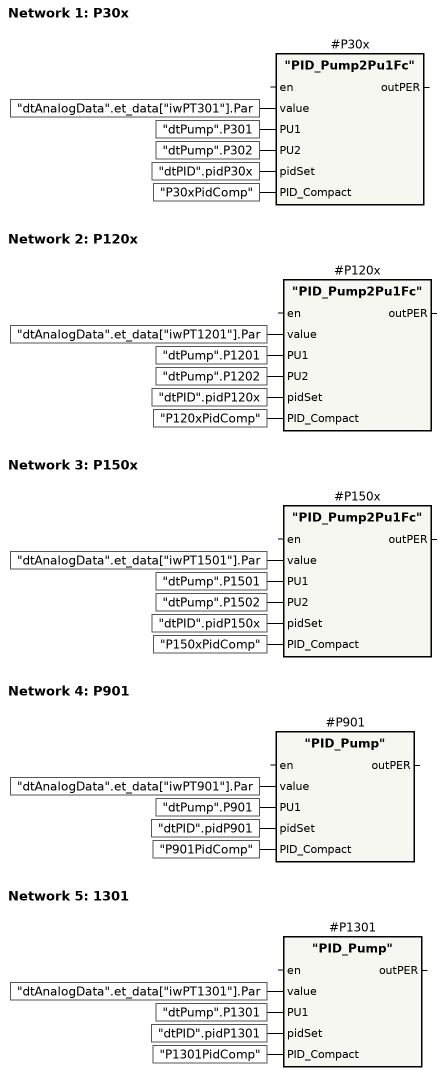
   #P30x(value := "dtAnalogData".et_data["iwPT301"].Par,   // "PID_Pump2Pu1Fc"
         PU1 := "dtPump".P301,
         PU2 := "dtPump".P302,
         pidSet := "dtPID".pidP30x,
         PID_Compact := "P30xPidComp");
END_REGION

REGION Network 2: P120x
   #P120x(value := "dtAnalogData".et_data["iwPT1201"].Par,   // "PID_Pump2Pu1Fc"
          PU1 := "dtPump".P1201,
          PU2 := "dtPump".P1202,
          pidSet := "dtPID".pidP120x,
          PID_Compact := "P120xPidComp");
END_REGION

REGION Network 3: P150x
   #P150x(value := "dtAnalogData".et_data["iwPT1501"].Par,   // "PID_Pump2Pu1Fc"
          PU1 := "dtPump".P1501,
          PU2 := "dtPump".P1502,
          pidSet := "dtPID".pidP150x,
          PID_Compact := "P150xPidComp");
END_REGION

REGION Network 4: P901
   #P901(value := "dtAnalogData".et_data["iwPT901"].Par,   // "PID_Pump"
         PU1 := "dtPump".P901,
         pidSet := "dtPID".pidP901,
         PID_Compact := "P901PidComp");
END_REGION

REGION Network 5: 1301
   #P1301(value := "dtAnalogData".et_data["iwPT1301"].Par,   // "PID_Pump"
          PU1 := "dtPump".P1301,
          pidSet := "dtPID".pidP1301,
          PID_Compact := "P1301PidComp");
END_REGION
END_FUNCTION_BLOCK

FUNCTION_BLOCK "PID_Pump2Pu1Fc"   // FB59, FBD
{ S7_Optimized_Access := 'TRUE' }
VERSION : 0.1
// stored: AutoNumber true, IsIECCheckEnabled false, IsRetainMemResEnabled false, MemoryReserve 100, SetENOAutomatically false, UDAEnableTagReadback false
   VAR_INPUT
      value : Real;
      PU1 : "Pump";
      PU2 : "Pump";
   END_VAR
   VAR_OUTPUT
      outPER : Int;
   END_VAR
   VAR_IN_OUT
      pidSet : "setPID";
      PID_Compact : PID_Compact;
   END_VAR
   VAR
      pTrigAutoMode : Bool;
      pTrigManualMode : Bool;
      pTrigCmAuto1 : Bool;
      pTrigCmAuto2 : Bool;
      nTrigCmAuto1 : Bool;
      nTrigCmAuto2 : Bool;
      pTrigFix : Bool;
      nTrigFix : Bool;
      pTrigFreez : Bool;
      nTrigFreez : Bool;
      pTrigCmHand : Bool;
      nTrigCmHand : Bool;
   END_VAR
   VAR_TEMP   // added for the SCL form of the ladder/FBD networks
      _w1 : Bool;
      _w2 : Bool;
      _w3 : Bool;
      _w4 : Bool;
      _w5 : Bool;
      _w6 : Bool;
      _w7 : Bool;
      _w8 : Bool;
      _w9 : Bool;
      _w10 : Bool;
   END_VAR
BEGIN

REGION Network 1: Интеграл
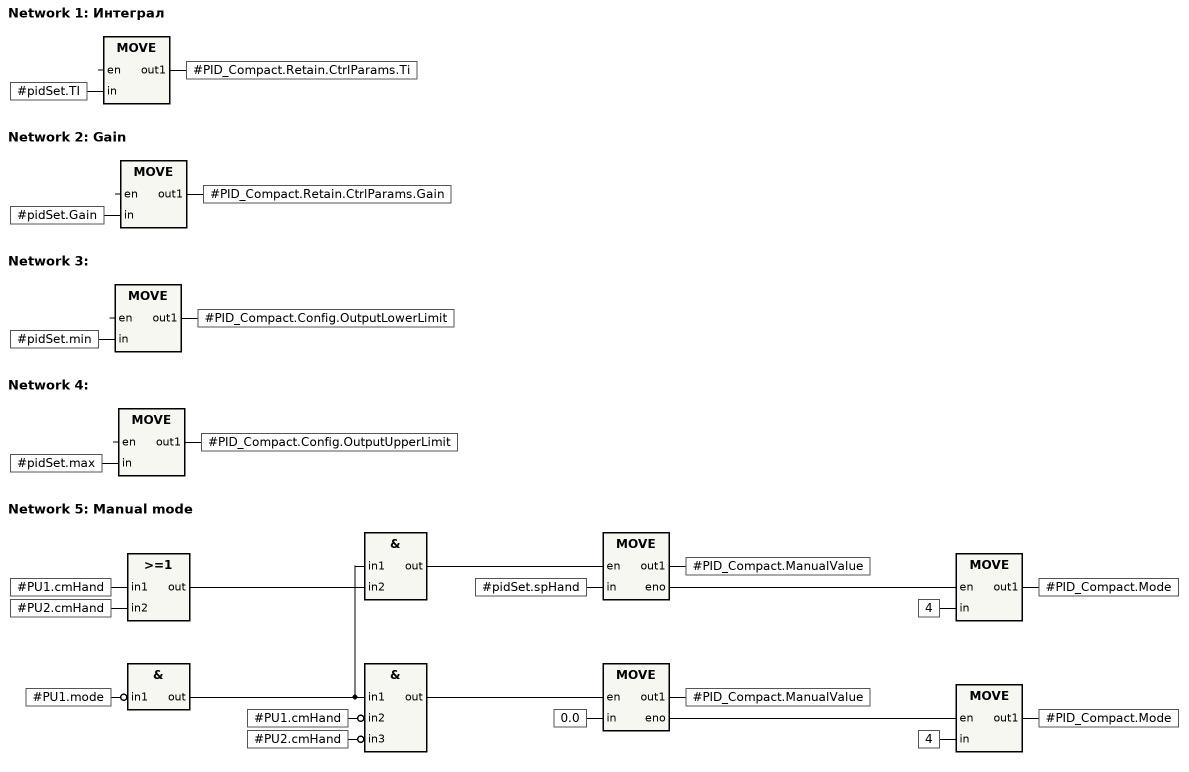
   #PID_Compact.Retain.CtrlParams.Ti := #pidSet.TI;
END_REGION

REGION Network 2: Gain
   #PID_Compact.Retain.CtrlParams.Gain := #pidSet.Gain;
END_REGION

REGION Network 3
   #PID_Compact.Config.OutputLowerLimit := #pidSet.min;
END_REGION

REGION Network 4
   #PID_Compact.Config.OutputUpperLimit := #pidSet.max;
END_REGION

REGION Network 5: Manual mode
   IF NOT #PU1.mode AND (#PU1.cmHand OR #PU2.cmHand) THEN
       #PID_Compact.ManualValue := #pidSet.spHand;
       #PID_Compact.Mode := 4;
   END_IF;
   IF NOT #PU1.mode AND NOT #PU1.cmHand AND NOT #PU2.cmHand THEN
       #PID_Compact.ManualValue := 0.0;
       #PID_Compact.Mode := 4;
   END_IF;
END_REGION

REGION Network 6: Auto mode
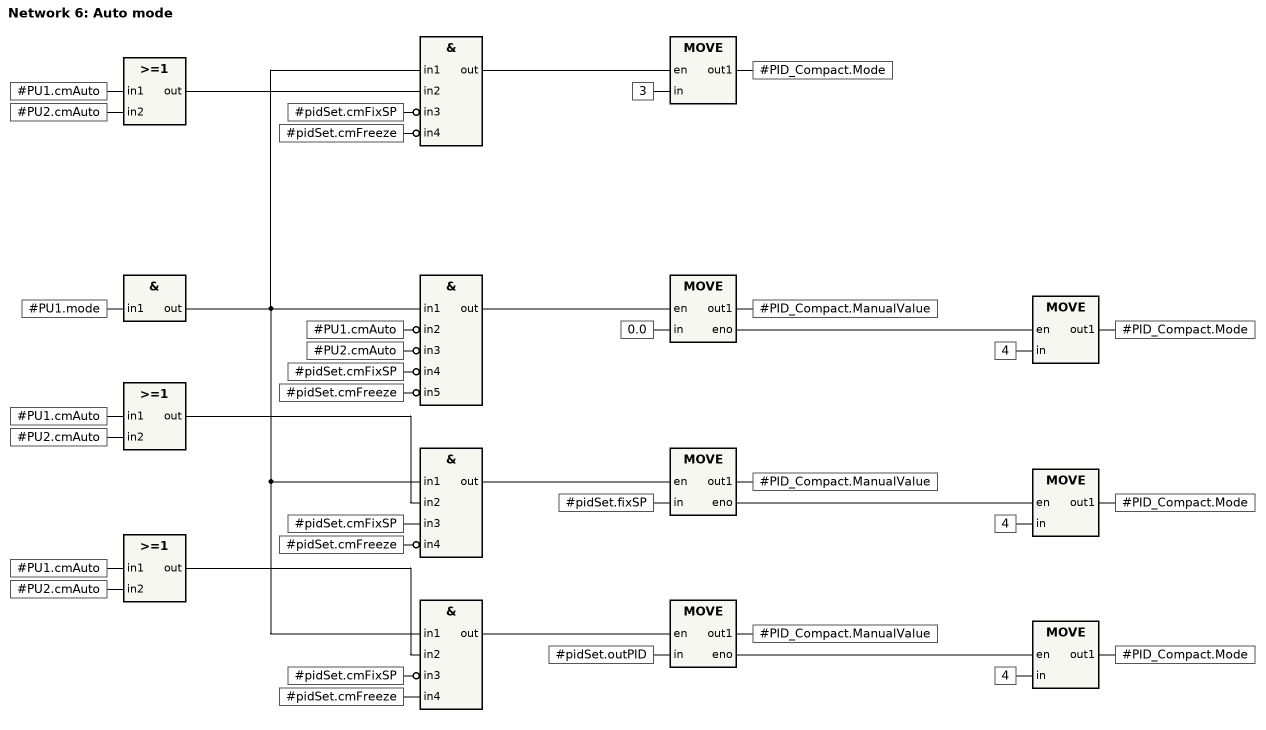
   IF #PU1.mode AND (#PU1.cmAuto OR #PU2.cmAuto) AND NOT #pidSet.cmFixSP AND NOT #pidSet.cmFreeze THEN
       #PID_Compact.Mode := 3;
   END_IF;
   IF #PU1.mode AND NOT #PU1.cmAuto AND NOT #PU2.cmAuto AND NOT #pidSet.cmFixSP AND NOT #pidSet.cmFreeze THEN
       #PID_Compact.ManualValue := 0.0;
       #PID_Compact.Mode := 4;
   END_IF;
   IF #PU1.mode AND (#PU1.cmAuto OR #PU2.cmAuto) AND #pidSet.cmFixSP AND NOT #pidSet.cmFreeze THEN
       #PID_Compact.ManualValue := #pidSet.fixSP;
       #PID_Compact.Mode := 4;
   END_IF;
   IF #PU1.mode AND (#PU1.cmAuto OR #PU2.cmAuto) AND NOT #pidSet.cmFixSP AND #pidSet.cmFreeze THEN
       #PID_Compact.ManualValue := #pidSet.outPID;
       #PID_Compact.Mode := 4;
   END_IF;
END_REGION

REGION Network 7: Set modeActivate
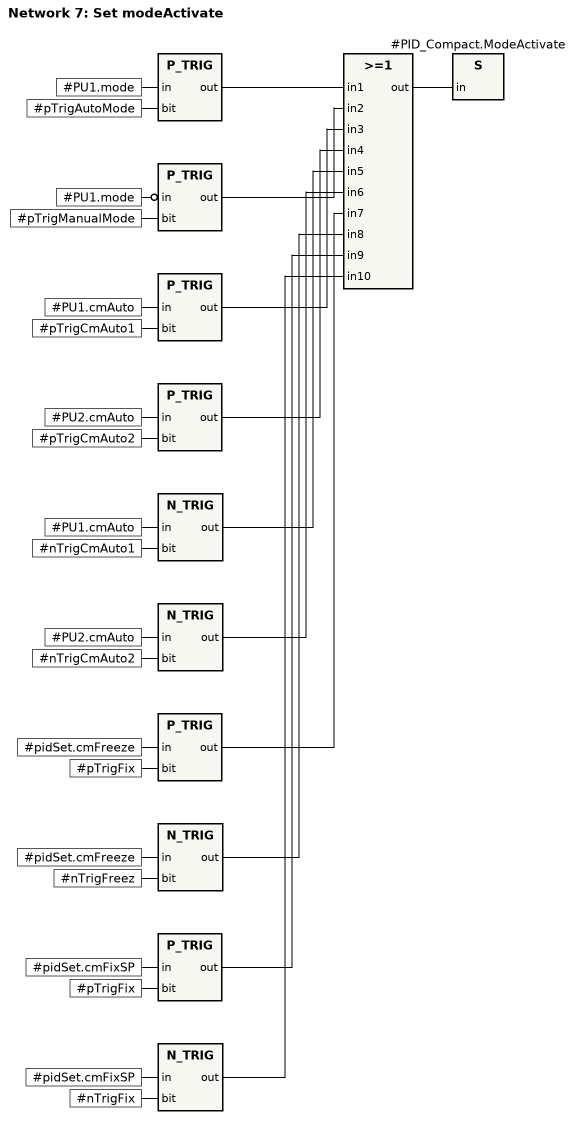
   #_w1 := #PU1.mode AND NOT #pTrigAutoMode;   // rising edge
   #pTrigAutoMode := #PU1.mode;
   #_w2 := NOT #PU1.mode AND NOT #pTrigManualMode;   // rising edge
   #pTrigManualMode := NOT #PU1.mode;
   #_w3 := #PU1.cmAuto AND NOT #pTrigCmAuto1;   // rising edge
   #pTrigCmAuto1 := #PU1.cmAuto;
   #_w4 := #PU2.cmAuto AND NOT #pTrigCmAuto2;   // rising edge
   #pTrigCmAuto2 := #PU2.cmAuto;
   #_w5 := NOT #PU1.cmAuto AND #nTrigCmAuto1;   // falling edge
   #nTrigCmAuto1 := #PU1.cmAuto;
   #_w6 := NOT #PU2.cmAuto AND #nTrigCmAuto2;   // falling edge
   #nTrigCmAuto2 := #PU2.cmAuto;
   #_w7 := #pidSet.cmFreeze AND NOT #pTrigFix;   // rising edge
   #pTrigFix := #pidSet.cmFreeze;
   #_w8 := NOT #pidSet.cmFreeze AND #nTrigFreez;   // falling edge
   #nTrigFreez := #pidSet.cmFreeze;
   #_w9 := #pidSet.cmFixSP AND NOT #pTrigFix;   // rising edge
   #pTrigFix := #pidSet.cmFixSP;
   #_w10 := NOT #pidSet.cmFixSP AND #nTrigFix;   // falling edge
   #nTrigFix := #pidSet.cmFixSP;
   IF #_w1 OR #_w2 OR #_w3 OR #_w4 OR #_w5 OR #_w6 OR #_w7 OR #_w8 OR #_w9 OR #_w10 THEN
       #PID_Compact.ModeActivate := TRUE;
   END_IF;
END_REGION

REGION Network 8
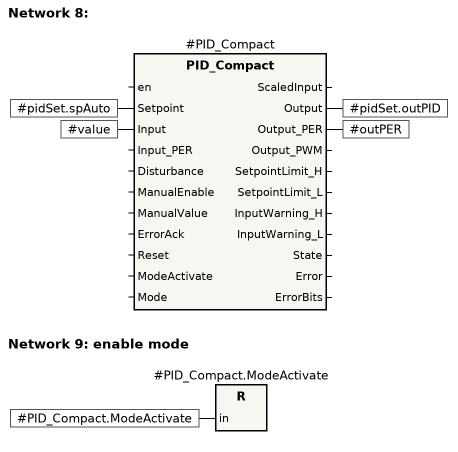
   #PID_Compact(Setpoint := #pidSet.spAuto, Input := #value, Output => #pidSet.outPID, Output_PER => #outPER);   // PID_Compact
END_REGION

REGION Network 9: enable mode
   IF #PID_Compact.ModeActivate THEN #PID_Compact.ModeActivate := FALSE; END_IF;
END_REGION
END_FUNCTION_BLOCK

FUNCTION_BLOCK "PID_Pump"   // FB62, FBD
{ S7_Optimized_Access := 'TRUE' }
VERSION : 0.1
// stored: AutoNumber false, IsIECCheckEnabled false, IsRetainMemResEnabled false, MemoryReserve 100, SetENOAutomatically false, UDAEnableTagReadback false
   VAR_INPUT
      value : Real;
      PU1 : "Pump";
   END_VAR
   VAR_OUTPUT
      outPER : Int;
   END_VAR
   VAR_IN_OUT
      pidSet : "setPID";
      PID_Compact : PID_Compact;
   END_VAR
   VAR
      pTrigAutoMode : Bool;
      pTrigManualMode : Bool;
      pTrigCmAuto1 : Bool;
      pTrigCmAuto2 : Bool;
      nTrigCmAuto1 : Bool;
      nTrigCmAuto2 : Bool;
      pTrigFix : Bool;
      nTrigFix : Bool;
      pTrigFreez : Bool;
      nTrigFreez : Bool;
      pTrigCmHand : Bool;
      nTrigCmHand : Bool;
   END_VAR
   VAR_TEMP   // added for the SCL form of the ladder/FBD networks
      _w1 : Bool;
      _w2 : Bool;
      _w3 : Bool;
      _w4 : Bool;
      _w5 : Bool;
      _w6 : Bool;
      _w7 : Bool;
      _w8 : Bool;
   END_VAR
BEGIN

REGION Network 1: Интеграл
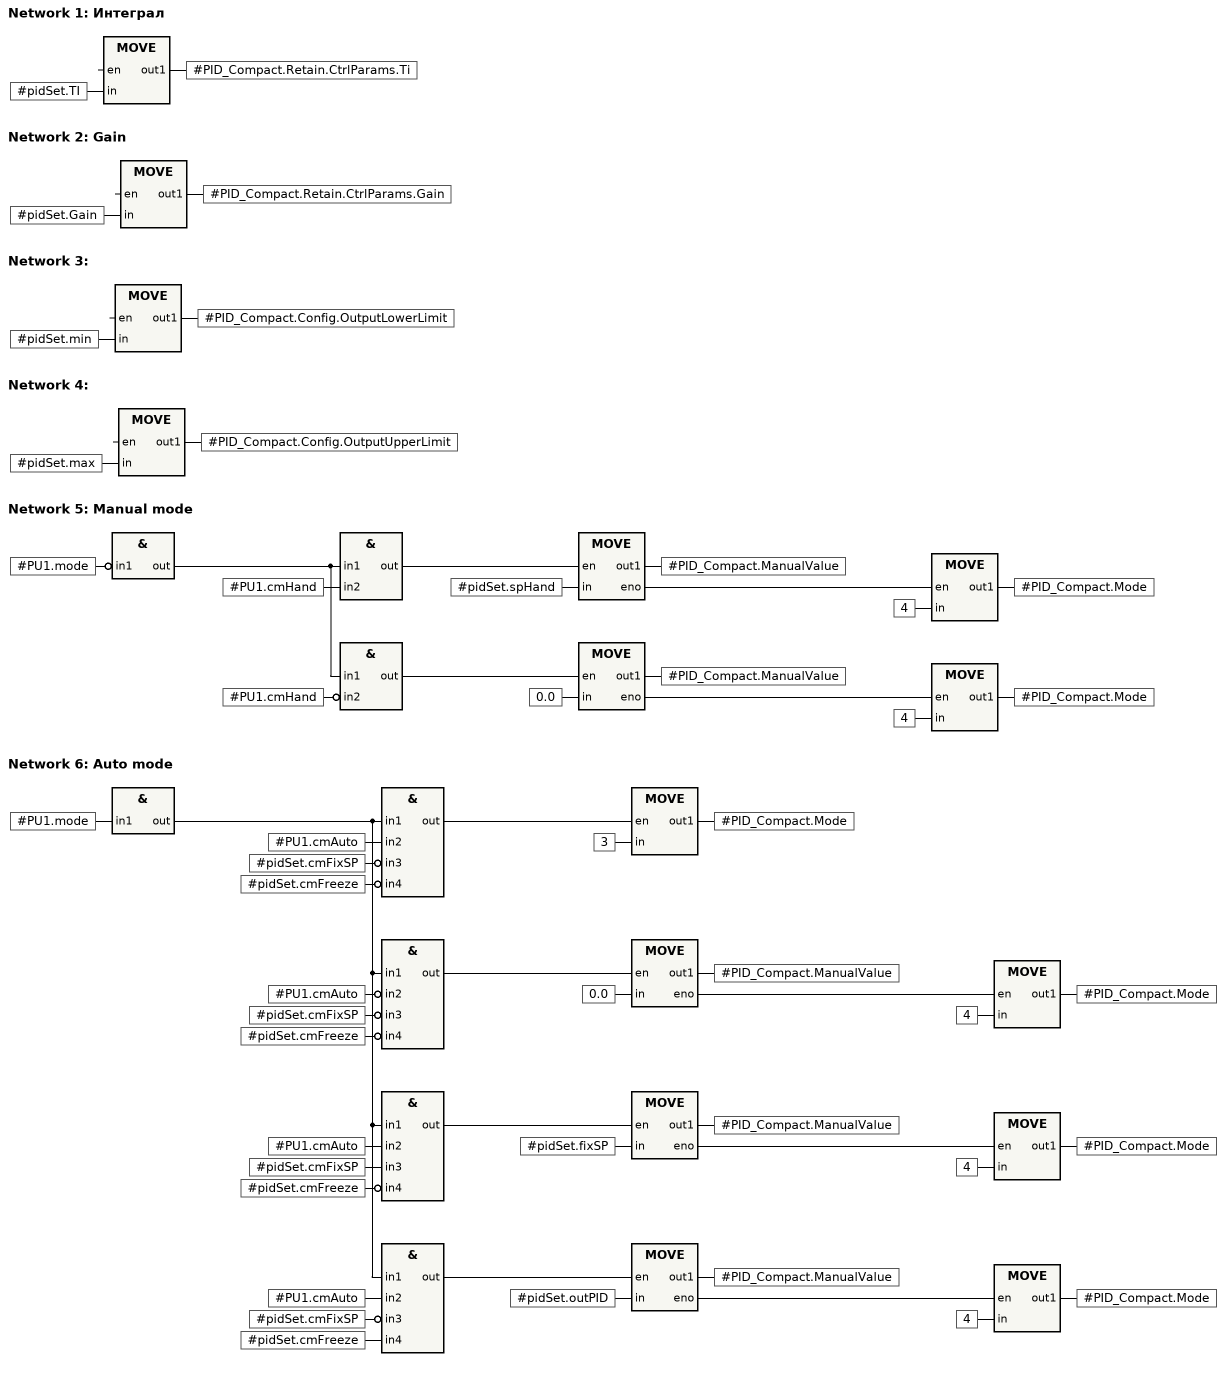
   #PID_Compact.Retain.CtrlParams.Ti := #pidSet.TI;
END_REGION

REGION Network 2: Gain
   #PID_Compact.Retain.CtrlParams.Gain := #pidSet.Gain;
END_REGION

REGION Network 3
   #PID_Compact.Config.OutputLowerLimit := #pidSet.min;
END_REGION

REGION Network 4
   #PID_Compact.Config.OutputUpperLimit := #pidSet.max;
END_REGION

REGION Network 5: Manual mode
   IF NOT #PU1.mode AND #PU1.cmHand THEN
       #PID_Compact.ManualValue := #pidSet.spHand;
       #PID_Compact.Mode := 4;
   END_IF;
   IF NOT #PU1.mode AND NOT #PU1.cmHand THEN
       #PID_Compact.ManualValue := 0.0;
       #PID_Compact.Mode := 4;
   END_IF;
END_REGION

REGION Network 6: Auto mode
   IF #PU1.mode AND #PU1.cmAuto AND NOT #pidSet.cmFixSP AND NOT #pidSet.cmFreeze THEN
       #PID_Compact.Mode := 3;
   END_IF;
   IF #PU1.mode AND NOT #PU1.cmAuto AND NOT #pidSet.cmFixSP AND NOT #pidSet.cmFreeze THEN
       #PID_Compact.ManualValue := 0.0;
       #PID_Compact.Mode := 4;
   END_IF;
   IF #PU1.mode AND #PU1.cmAuto AND #pidSet.cmFixSP AND NOT #pidSet.cmFreeze THEN
       #PID_Compact.ManualValue := #pidSet.fixSP;
       #PID_Compact.Mode := 4;
   END_IF;
   IF #PU1.mode AND #PU1.cmAuto AND NOT #pidSet.cmFixSP AND #pidSet.cmFreeze THEN
       #PID_Compact.ManualValue := #pidSet.outPID;
       #PID_Compact.Mode := 4;
   END_IF;
END_REGION

REGION Network 7: Set modeActivate
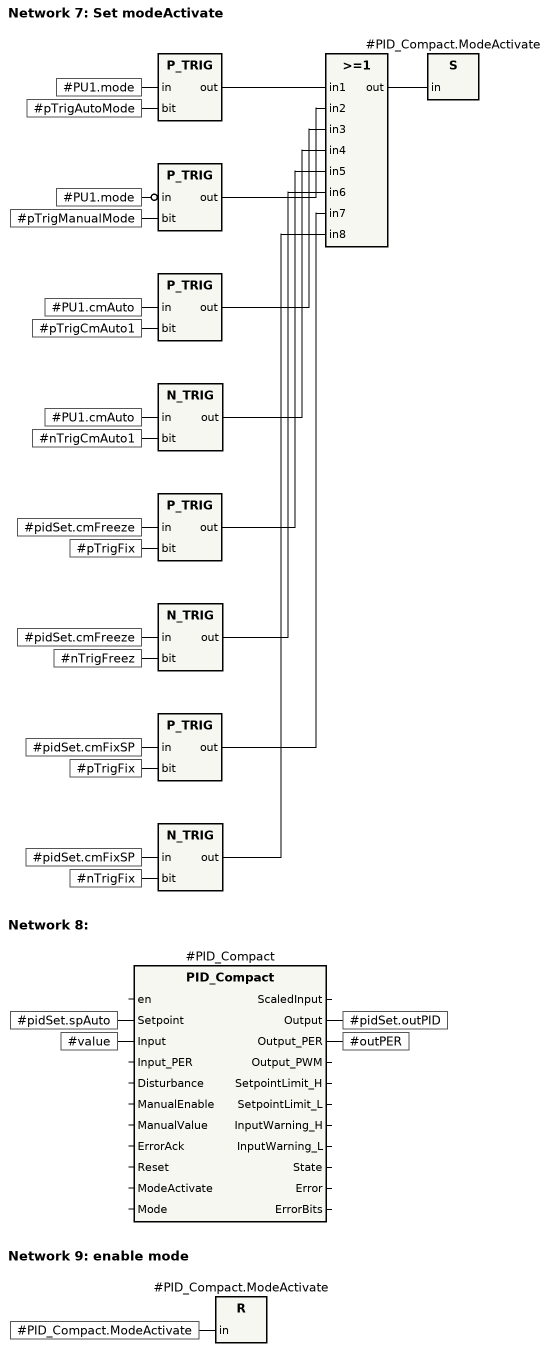
   #_w1 := #PU1.mode AND NOT #pTrigAutoMode;   // rising edge
   #pTrigAutoMode := #PU1.mode;
   #_w2 := NOT #PU1.mode AND NOT #pTrigManualMode;   // rising edge
   #pTrigManualMode := NOT #PU1.mode;
   #_w3 := #PU1.cmAuto AND NOT #pTrigCmAuto1;   // rising edge
   #pTrigCmAuto1 := #PU1.cmAuto;
   #_w4 := NOT #PU1.cmAuto AND #nTrigCmAuto1;   // falling edge
   #nTrigCmAuto1 := #PU1.cmAuto;
   #_w5 := #pidSet.cmFreeze AND NOT #pTrigFix;   // rising edge
   #pTrigFix := #pidSet.cmFreeze;
   #_w6 := NOT #pidSet.cmFreeze AND #nTrigFreez;   // falling edge
   #nTrigFreez := #pidSet.cmFreeze;
   #_w7 := #pidSet.cmFixSP AND NOT #pTrigFix;   // rising edge
   #pTrigFix := #pidSet.cmFixSP;
   #_w8 := NOT #pidSet.cmFixSP AND #nTrigFix;   // falling edge
   #nTrigFix := #pidSet.cmFixSP;
   IF #_w1 OR #_w2 OR #_w3 OR #_w4 OR #_w5 OR #_w6 OR #_w7 OR #_w8 THEN
       #PID_Compact.ModeActivate := TRUE;
   END_IF;
END_REGION

REGION Network 8
   #PID_Compact(Setpoint := #pidSet.spAuto, Input := #value, Output => #pidSet.outPID, Output_PER => #outPER);   // PID_Compact
END_REGION

REGION Network 9: enable mode
   IF #PID_Compact.ModeActivate THEN #PID_Compact.ModeActivate := FALSE; END_IF;
END_REGION
END_FUNCTION_BLOCK

FUNCTION_BLOCK "TONR_200ms"   // FB10, FBD
{ S7_Optimized_Access := 'TRUE' }
VERSION : 0.1
// stored: AutoNumber true, IsIECCheckEnabled false, IsRetainMemResEnabled false, MemoryReserve 100, SetENOAutomatically false, UDAEnableTagReadback false
   VAR_INPUT
      In : Bool;
      PT : Time;
      R : Bool;
   END_VAR
   VAR_OUTPUT
      ET : Time;
      Q : Bool;
   END_VAR
BEGIN

REGION Network 1: Увеличение текущего времени
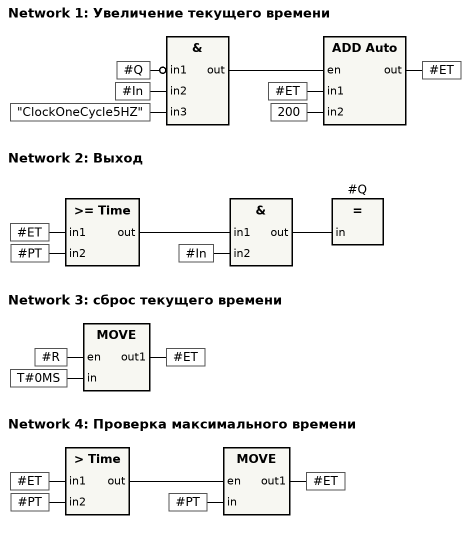
   IF NOT #Q AND #In AND "ClockOneCycle5HZ" THEN #ET := #ET + 200; END_IF;
END_REGION

REGION Network 2: Выход
   #Q := (#ET >= #PT) AND #In;
END_REGION

REGION Network 3: сброс текущего времени
   IF #R THEN #ET := T#0MS; END_IF;
END_REGION

REGION Network 4: Проверка максимального времени
   IF #ET > #PT THEN #ET := #PT; END_IF;
END_REGION
END_FUNCTION_BLOCK

FUNCTION_BLOCK "TON_200ms"   // FB9, FBD
{ S7_Optimized_Access := 'TRUE' }
VERSION : 0.1
// stored: AutoNumber true, IsIECCheckEnabled false, IsRetainMemResEnabled false, MemoryReserve 100, SetENOAutomatically false, UDAEnableTagReadback false
   VAR_INPUT
      In : Bool;
      PT : Time;
   END_VAR
   VAR_OUTPUT
      ET : Time;
      Q : Bool;
   END_VAR
BEGIN

REGION Network 1: Увеличение текущего времени
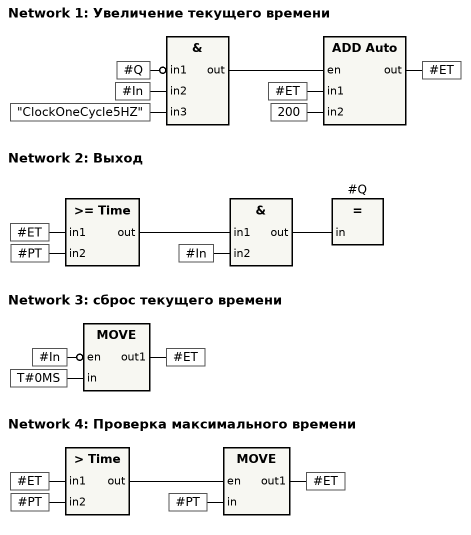
   IF NOT #Q AND #In AND "ClockOneCycle5HZ" THEN #ET := #ET + 200; END_IF;
END_REGION

REGION Network 2: Выход
   #Q := (#ET >= #PT) AND #In;
END_REGION

REGION Network 3: сброс текущего времени
   IF NOT #In THEN #ET := T#0MS; END_IF;
END_REGION

REGION Network 4: Проверка максимального времени
   IF #ET > #PT THEN #ET := #PT; END_IF;
END_REGION
END_FUNCTION_BLOCK

FUNCTION "setFlags" : Void   // FC2, FBD
{ S7_Optimized_Access := 'TRUE' }
VERSION : 0.1
// stored: AutoNumber true, IsIECCheckEnabled false, SetENOAutomatically false, UDAEnableTagReadback false
   VAR_INPUT
      enCondition : Bool;
      condition : Bool;
      setTimerVal : Real;
   END_VAR
   VAR_IN_OUT
      curFlag : Bool;
      mainFlag : Bool;
      timerVal : Real;
   END_VAR
BEGIN

REGION Network 1 (SCL)

   #curFlag := #enCondition AND #condition;

   IF NOT #curFlag THEN
       #timerVal := 0;
   END_IF;

   IF #curFlag AND #timerVal < #setTimerVal THEN
       #timerVal += 0.1;
   END_IF;

   IF #timerVal >= #setTimerVal THEN
       #mainFlag := TRUE;
   END_IF;
END_REGION
END_FUNCTION

FUNCTION "setState" : Void   // FC3, FBD
{ S7_Optimized_Access := 'TRUE' }
VERSION : 0.1
// stored: AutoNumber true, IsIECCheckEnabled false, SetENOAutomatically false, UDAEnableTagReadback false
   VAR_INPUT
      condition : Bool;
      hexVal : Word;
   END_VAR
   VAR_IN_OUT
      state : Word;
   END_VAR
BEGIN

REGION Network 1 (SCL)
   IF #condition THEN
       // Statement section IF
       #state := #state OR #hexVal;
   ELSE
       #state := #state AND NOT #hexVal;
   END_IF;
END_REGION
END_FUNCTION

FUNCTION_BLOCK "DPumpCntr"   // FB70, LAD
{ S7_Optimized_Access := 'FALSE' }
VERSION : 0.1
// #ST:
// номер бита, часло десятичное
//  0  - стоп 
// 0 1 - работа
// 1 2 - запуск
// 2 4 - остановка
// 3 8 - сервисный режим
// 4 16 - ошибка Пуска
// 5 32 - ошибка Стопа
// 6 64 - ошибка питания
// 7 128 - ошибка частотника (дозатора)
// 8 256 - Блокировка внешняя
// 9 - 512 - нажат аварийный стоп
// 10 -1024 - сборная авария
// 11 2048
// 12 4096
// 13 8192
// 14 16384 
// 15 32768 - режим 0-ручной, 1-авто
// 
// показывать кнопки ручного управления
// stored: AutoNumber false, IsIECCheckEnabled false, SetENOAutomatically false, UDAEnableTagReadback false
   VAR_INPUT
      power : Bool;   // питание устройства
      run : Bool;
      emrStop : Bool;   // Авариный стоп 0-авария, 1-ок
      alarmFC : Bool;   // 1-авария
      Ack : Bool;   // Сброс Аварий
      FE : Real;
   END_VAR
   VAR_OUTPUT
      qStart : Bool;
      pqw : Int;
   END_VAR
   VAR_IN_OUT
      dev : "DPump";
      prop : "PropDosing";
   END_VAR
   VAR DB_SPECIFIC
      ErrOC : Bool;   // Признак аварии по закрытию или открытию
      ErrPower : Bool;   // Признак аварии питания
      ErrDis : Bool;   // Признак внешней блокировки
      qON : Bool;   // Выход для управления механизмом
      tmrClosing { S7_SetPoint := 'True'} : TON_TIME;
      tmrOpening { S7_SetPoint := 'True'} : TON_TIME;
      closed : Bool;
      opened : Bool;
      closing : Bool;
      opening : Bool;
      errStart : Bool;
      errStop : Bool;
      errEmrStop : Bool;
      errAlarmFc : Bool;
      errService : Bool;
      tStart : Time;
      tStop : Time;
   END_VAR
   VAR
      ServiceEventHandler { S7_SetPoint := 'True'} : "DevAckSingleAlarm";
      PowerEventHandler { S7_SetPoint := 'True'} : "DevAckSingleAlarm";
      DevAlarmEventHandler { S7_SetPoint := 'True'} : "DevAckSingleAlarm";
      DisEventHandler { S7_SetPoint := 'True'} : "DevAckSingleAlarm";
      EmrStopEventHandler { S7_SetPoint := 'True'} : "DevAckSingleAlarm";
      BadStartEventHandler { S7_SetPoint := 'True'} : "DevAckSingleAlarm";
      BadStopEventHandler { S7_SetPoint := 'True'} : "DevAckSingleAlarm";
   END_VAR
BEGIN

REGION Network 1: Сброс состояния
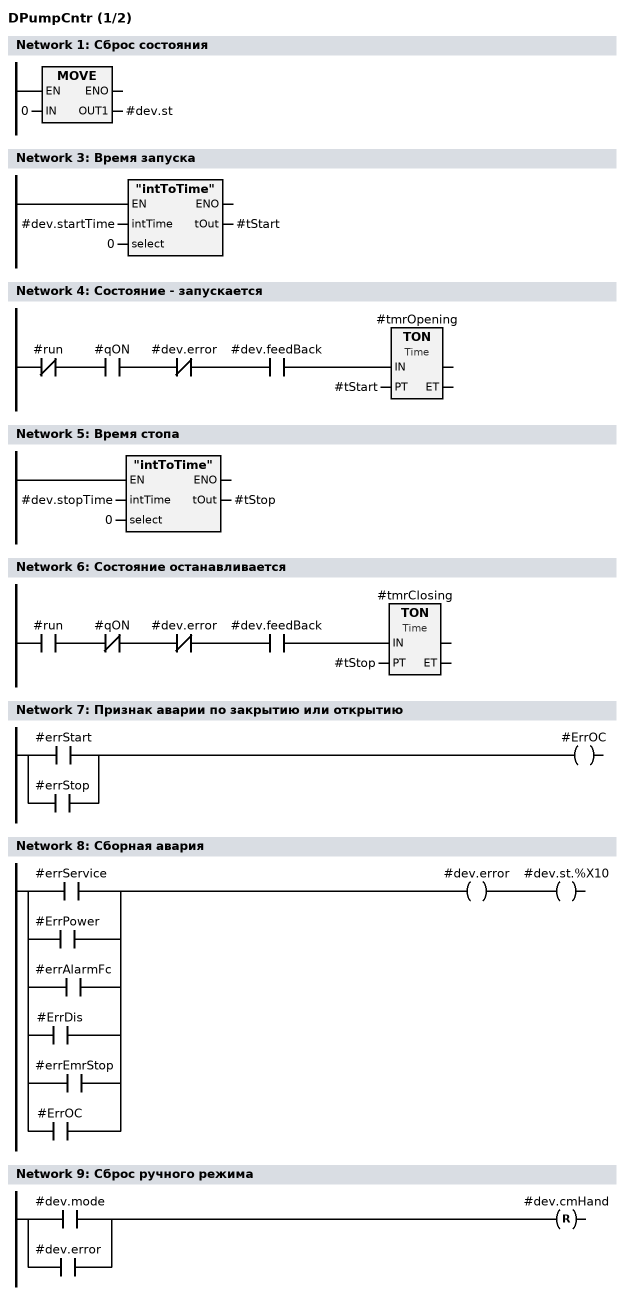
   RUNG wire#powerrail
      { S7_GenerateENO := "TRUE" } Move(in := 0, out1 => #dev.st)
   END_RUNG
   // the same network as SCL:
   #dev.st := 0;
END_REGION

REGION Network 2 (SCL): Event handlers
   #ServiceEventHandler(alarmSignal := #dev.service,
                        ack := #Ack,
                        ackBit := #dev.ack.%X3,
                        stateBit := #dev.st.%X3,
                        alarmTag := #errService);
   #BadStartEventHandler(alarmSignal:=#tmrOpening.Q,
                         ack:=#Ack,
                         ackBit:=#dev.ack.%X4,
                         stateBit:=#dev.st.%X4,
                         alarmTag:=#errStart);
   #BadStopEventHandler(alarmSignal:=#tmrClosing.Q,
                        ack:=#Ack,
                        ackBit:=#dev.ack.%X5,
                        stateBit:=#dev.ack.%X5,
                        alarmTag:=#errStop);
   #PowerEventHandler(alarmSignal := #power,
                      ack := #Ack,
                      ackBit := #dev.ack.%X6,
                      stateBit := #dev.st.%X6,
                      alarmTag := #ErrPower);
   #DevAlarmEventHandler(alarmSignal := #alarmFC,
                         ack := #Ack,
                         ackBit := #dev.ack.%X7,
                         stateBit := #dev.st.%X7,
                         alarmTag := #errAlarmFc);
   #DisEventHandler(alarmSignal := #dev.block,
                    ack := #Ack,
                    ackBit := #dev.ack.%X8,
                    stateBit := #dev.st.%X8,
                    alarmTag := #ErrDis);
   #EmrStopEventHandler(alarmSignal := #emrStop,
                        ack := #Ack,
                        ackBit := #dev.ack.%X9,
                        stateBit := #dev.st.%X9,
                        alarmTag := #errEmrStop);
END_REGION

REGION Network 3: Время запуска
   RUNG wire#powerrail
      "intToTime"(intTime := #dev.startTime, select := 0, tOut => #tStart)
   END_RUNG
   // the same network as SCL:
   "intToTime"(intTime := #dev.startTime, select := 0, tOut => #tStart);
END_REGION

REGION Network 4: Состояние - запускается
   RUNG wire#powerrail
      I_Contact( #run )
      Contact( #qON )
      I_Contact( #dev.error )
      Contact( #dev.feedBack )
      { S7_Templates := "time_type := Time" } #tmrOpening.TON(pt := #tStart, et =>)
   END_RUNG
   // the same network as SCL:
   #tmrOpening(IN := NOT #run AND #qON AND NOT #dev.error AND #dev.feedBack, PT := #tStart);   // TON
END_REGION

REGION Network 5: Время стопа
   RUNG wire#powerrail
      "intToTime"(intTime := #dev.stopTime, select := 0, tOut => #tStop)
   END_RUNG
   // the same network as SCL:
   "intToTime"(intTime := #dev.stopTime, select := 0, tOut => #tStop);
END_REGION

REGION Network 6: Состояние останавливается
   RUNG wire#powerrail
      Contact( #run )
      I_Contact( #qON )
      I_Contact( #dev.error )
      Contact( #dev.feedBack )
      { S7_Templates := "time_type := Time" } #tmrClosing.TON(pt := #tStop, et =>)
   END_RUNG
   // the same network as SCL:
   #tmrClosing(IN := #run AND NOT #qON AND NOT #dev.error AND #dev.feedBack, PT := #tStop);   // TON
END_REGION

REGION Network 7: Признак аварии по закрытию или открытию
   RUNG wire#powerrail
      Contact( #errStart )
      wire#w1
      Coil( #ErrOC )
   END_RUNG
   RUNG wire#powerrail
      Contact( #errStop )
   END_RUNG wire#w1
   // the same network as SCL:
   #ErrOC := #errStart OR #errStop;
END_REGION

REGION Network 8: Сборная авария
   RUNG wire#powerrail
      Contact( #errService )
      wire#w1
      Coil( #dev.error )
      Coil( #dev.st.%X10 )
   END_RUNG
   RUNG wire#powerrail
      Contact( #ErrPower )
   END_RUNG wire#w1
   RUNG wire#powerrail
      Contact( #errAlarmFc )
   END_RUNG wire#w1
   RUNG wire#powerrail
      Contact( #ErrDis )
   END_RUNG wire#w1
   RUNG wire#powerrail
      Contact( #errEmrStop )
   END_RUNG wire#w1
   RUNG wire#powerrail
      Contact( #ErrOC )
   END_RUNG wire#w1
   // the same network as SCL:
   #dev.error := #errService OR #ErrPower OR #errAlarmFc OR #ErrDis OR #errEmrStop OR #ErrOC;
   #dev.st.%X10 := #dev.error;
END_REGION

REGION Network 9: Сброс ручного режима
   RUNG wire#powerrail
      Contact( #dev.mode )
      wire#w1
      R_Coil( #dev.cmHand )
   END_RUNG
   RUNG wire#powerrail
      Contact( #dev.error )
   END_RUNG wire#w1
   // the same network as SCL:
   IF #dev.mode OR #dev.error THEN #dev.cmHand := FALSE; END_IF;
END_REGION

REGION Network 10: Сброс авто режима
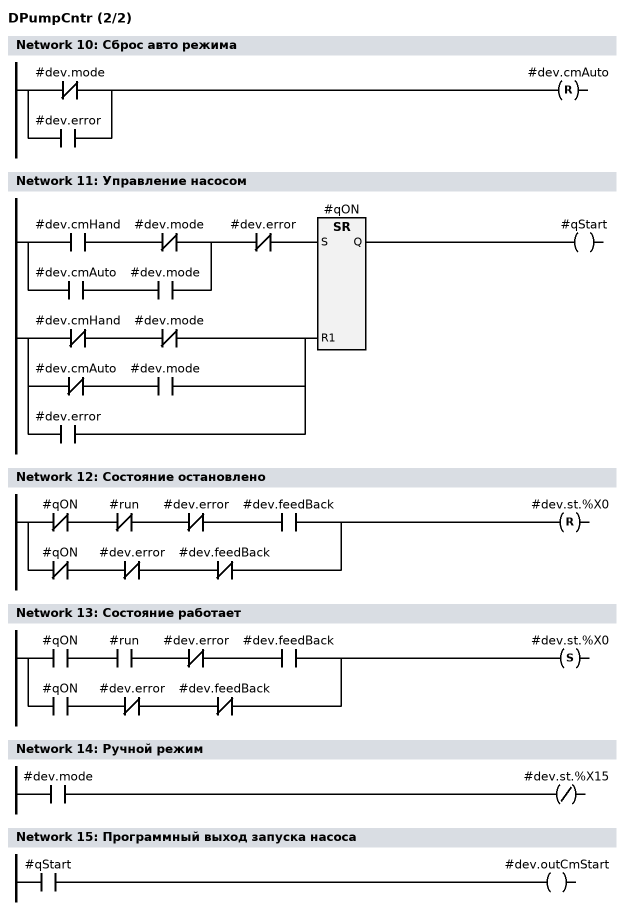
   RUNG wire#powerrail
      I_Contact( #dev.mode )
      wire#w1
      R_Coil( #dev.cmAuto )
   END_RUNG
   RUNG wire#powerrail
      Contact( #dev.error )
   END_RUNG wire#w1
   // the same network as SCL:
   IF NOT #dev.mode OR #dev.error THEN #dev.cmAuto := FALSE; END_IF;
END_REGION

REGION Network 11: Управление насосом
   RUNG wire#powerrail
      Contact( #dev.cmHand )
      I_Contact( #dev.mode )
      wire#w1
      I_Contact( #dev.error )
      S_SR(operand := #qON, r1 := wire#w2)
      Coil( #qStart )
   END_RUNG
   RUNG wire#powerrail
      Contact( #dev.cmAuto )
      Contact( #dev.mode )
   END_RUNG wire#w1
   RUNG wire#powerrail
      I_Contact( #dev.cmHand )
      I_Contact( #dev.mode )
   END_RUNG wire#w2
   RUNG wire#powerrail
      I_Contact( #dev.cmAuto )
      Contact( #dev.mode )
   END_RUNG wire#w2
   RUNG wire#powerrail
      Contact( #dev.error )
   END_RUNG wire#w2
   // the same network as SCL:
   IF ((#dev.cmHand AND NOT #dev.mode) OR (#dev.cmAuto AND #dev.mode)) AND NOT #dev.error THEN
       #qON := TRUE;   // SR flip-flop
   END_IF;
   IF (NOT #dev.cmHand AND NOT #dev.mode) OR (NOT #dev.cmAuto AND #dev.mode) OR #dev.error THEN
       #qON := FALSE;
   END_IF;
   #qStart := #qON;
END_REGION

REGION Network 12: Состояние остановлено
   RUNG wire#powerrail
      I_Contact( #qON )
      I_Contact( #run )
      I_Contact( #dev.error )
      Contact( #dev.feedBack )
      wire#w1
      R_Coil( #dev.st.%X0 )
   END_RUNG
   RUNG wire#powerrail
      I_Contact( #qON )
      I_Contact( #dev.error )
      I_Contact( #dev.feedBack )
   END_RUNG wire#w1
   // the same network as SCL:
   IF (NOT #qON AND NOT #run AND NOT #dev.error AND #dev.feedBack) OR (NOT #qON AND NOT #dev.error AND NOT #dev.feedBack) THEN
       #dev.st.%X0 := FALSE;
   END_IF;
END_REGION

REGION Network 13: Состояние работает
   RUNG wire#powerrail
      Contact( #qON )
      Contact( #run )
      I_Contact( #dev.error )
      Contact( #dev.feedBack )
      wire#w1
      S_Coil( #dev.st.%X0 )
   END_RUNG
   RUNG wire#powerrail
      Contact( #qON )
      I_Contact( #dev.error )
      I_Contact( #dev.feedBack )
   END_RUNG wire#w1
   // the same network as SCL:
   IF (#qON AND #run AND NOT #dev.error AND #dev.feedBack) OR (#qON AND NOT #dev.error AND NOT #dev.feedBack) THEN
       #dev.st.%X0 := TRUE;
   END_IF;
END_REGION

REGION Network 14: Ручной режим
   RUNG wire#powerrail
      Contact( #dev.mode )
      I_Coil( #dev.st.%X15 )
   END_RUNG
   // the same network as SCL:
   #dev.st.%X15 := NOT #dev.mode;
END_REGION

REGION Network 15: Программный выход запуска насоса
   RUNG wire#powerrail
      Contact( #qStart )
      Coil( #dev.outCmStart )
   END_RUNG
   // the same network as SCL:
   #dev.outCmStart := #qStart;
END_REGION

REGION Network 16 (SCL): Prop dossing
   //дозирование пропорционально расходу

   //производителньность л/ч

   IF #dev.mode AND #dev.cmAuto THEN
       //KVA
       IF #prop.enableFix THEN
           IF #prop.fixSP > 100 THEN
               #prop.fixSP := 100;
           END_IF;
           IF #prop.fixSP < 0 THEN
               #prop.fixSP := 0;
           END_IF;
           #prop.outLPH := (#prop.max * #prop.fixSP) / 100;
           //
           // #prop.outLPH := #prop.fixSP;
       ELSE
           IF #prop.density > 0 THEN
               #prop.outLPH := #FE * #prop.spAuto / (#prop.density * 1000.0);
           ELSE
               #prop.outLPH := 0;
           END_IF;

           //запрет дозирования если расход меньше заданного
           IF #FE < #prop.minFE THEN
               #prop.outLPH := 0.0;
           END_IF;
       END_IF;
   END_IF;
   IF NOT #dev.mode AND #dev.cmHand THEN
       #prop.outLPH := #prop.spHand;
   END_IF;

   //запрет дозирования
   IF NOT #dev.cmHand AND NOT #dev.cmAuto THEN
       #prop.outLPH := 0.0;
   END_IF;

   IF #prop.outLPH > #prop.max THEN
       #prop.outLPH := #prop.max;
   END_IF;

   //расчет PQW
   IF #prop.max > 0 THEN
       #pqw := REAL_TO_INT(#prop.outLPH * 27648.0 / #prop.max);
   ELSE
       #pqw := 0;
   END_IF;

   //ограничение выхода
   IF #pqw < 0 THEN
       #pqw := 0;
   END_IF;
   IF #pqw > 27648 THEN
       #pqw := 27648;
   END_IF;

   //расчет тока
   #prop.outmA := 4.0 + INT_TO_REAL(#pqw) * 16.0 / 27648.0;
   #prop.outSP := INT_TO_REAL(#pqw) * 100.0 / 27648.0;
   #prop.FE := #FE;
END_REGION
END_FUNCTION_BLOCK

FUNCTION_BLOCK "AvAckAlarm"   // FB48, LAD
{ S7_Optimized_Access := 'TRUE' }
VERSION : 0.1
// stored: AutoNumber true, IsIECCheckEnabled false, IsRetainMemResEnabled false, MemoryReserve 100, SetENOAutomatically false, UDAEnableTagReadback false
   VAR_INPUT
      ack : Bool;
      power : Bool;
      alarmFC : Bool;
      emrStop : Bool;   // Авариный стоп 0-авария, 1-ок
      local : Bool;   // 1-местный режим
      tmrOpening_Q : Bool;
      tmrClosing_Q : Bool;
   END_VAR
   VAR_IN_OUT
      dev : "Av";
      errService : Bool;
      ErrPower : Bool;   // Признак аварии питания
      errAlarmFc : Bool;
      ErrDis : Bool;   // Признак внешней блокировки
      errEmrStop : Bool;
      errLocal : Bool;
      errStart : Bool;
      errStop : Bool;
   END_VAR
   VAR
      InstService { S7_SetPoint := 'True'} : "DevAckSingleAlarm";
      InstPower { S7_SetPoint := 'True'} : "DevAckSingleAlarm";
      InstFc { S7_SetPoint := 'True'} : "DevAckSingleAlarm";
      InstDis { S7_SetPoint := 'True'} : "DevBlockAckSingleAlarm";
      InstEmrStop { S7_SetPoint := 'True'} : "DevAckSingleAlarm";
      InstLocal { S7_SetPoint := 'True'} : "DevAckSingleAlarm";
      InstStart { S7_SetPoint := 'True'} : "DevAckSingleAlarm";
      InstStop { S7_SetPoint := 'True'} : "DevAckSingleAlarm";
   END_VAR
BEGIN

REGION Network 1: Ошибка питания - нужно квитирование ACK
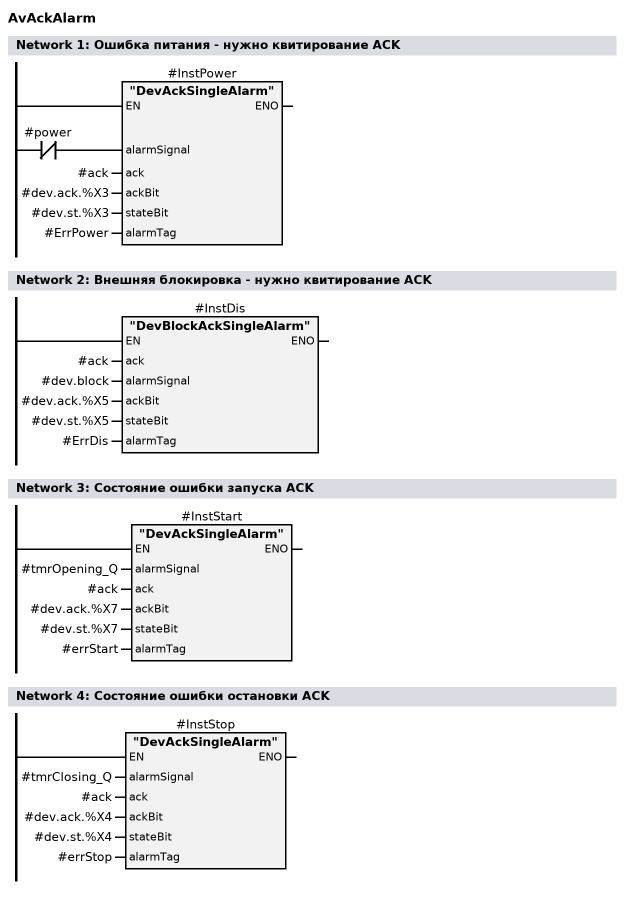
   RUNG wire#powerrail
      #InstPower(alarmSignal := wire#w1, ack := #ack, ackBit := #dev.ack.%X3, stateBit := #dev.st.%X3, alarmTag := #ErrPower)
   END_RUNG
   RUNG wire#powerrail
      I_Contact( #power )
   END_RUNG wire#w1
   // the same network as SCL:
   #InstPower(alarmSignal := NOT #power,   // "DevAckSingleAlarm"
              ack := #ack,
              ackBit := #dev.ack.%X3,
              stateBit := #dev.st.%X3,
              alarmTag := #ErrPower);
END_REGION

REGION Network 2: Внешняя блокировка - нужно квитирование ACK
   RUNG wire#powerrail
      #InstDis(ack := #ack, alarmSignal := #dev.block, ackBit := #dev.ack.%X5, stateBit := #dev.st.%X5, alarmTag := #ErrDis)
   END_RUNG
   // the same network as SCL:
   #InstDis(ack := #ack,   // "DevBlockAckSingleAlarm"
            alarmSignal := #dev.block,
            ackBit := #dev.ack.%X5,
            stateBit := #dev.st.%X5,
            alarmTag := #ErrDis);
END_REGION

REGION Network 3: Состояние ошибки запуска ACK
   RUNG wire#powerrail
      #InstStart(alarmSignal := #tmrOpening_Q, ack := #ack, ackBit := #dev.ack.%X7, stateBit := #dev.st.%X7, alarmTag := #errStart)
   END_RUNG
   // the same network as SCL:
   #InstStart(alarmSignal := #tmrOpening_Q,   // "DevAckSingleAlarm"
              ack := #ack,
              ackBit := #dev.ack.%X7,
              stateBit := #dev.st.%X7,
              alarmTag := #errStart);
END_REGION

REGION Network 4: Состояние ошибки остановки ACK
   RUNG wire#powerrail
      #InstStop(alarmSignal := #tmrClosing_Q, ack := #ack, ackBit := #dev.ack.%X4, stateBit := #dev.st.%X4, alarmTag := #errStop)
   END_RUNG
   // the same network as SCL:
   #InstStop(alarmSignal := #tmrClosing_Q,   // "DevAckSingleAlarm"
             ack := #ack,
             ackBit := #dev.ack.%X4,
             stateBit := #dev.st.%X4,
             alarmTag := #errStop);
END_REGION
END_FUNCTION_BLOCK

FUNCTION_BLOCK "AvCntrl"   // FB81, LAD
{ S7_Optimized_Access := 'FALSE' }
VERSION : 0.1
// #ST:
// 0 0 - закрыта - стоп 
// 1 1- открыта - работа
// 2 2 -открывается - запускается
// 3 4 -закрывается - останавливается 
// 4 8 - ошибка питания
// 5 16 - ошибка концевиков - закрытия
// 6 32 - Блокировка
// 7 64 - сборная авария
// 8 128 - ошибка концевиков - открытия
// 9 256 - не выбран режим
// 10 - 512 - показывать кнопки ручного управления
// 
// БИТ 13 - РЕЖИМ
// бит 14 - состояние концевиков - открыто
// 15 - закрыто
// stored: AutoNumber false, IsIECCheckEnabled true, SetENOAutomatically false, UDAEnableTagReadback false
   VAR_INPUT
      power : Bool;   // питание устройства
      open : Bool;   // Задвижка открыта
      close : Bool;   // Задвижка закрыта
   END_VAR
   VAR_OUTPUT
      qKm : Bool;   // Выход на управление механизмом 0-стоп, 1-пуск
   END_VAR
   VAR_IN_OUT
      dev : "Av";
   END_VAR
   VAR DB_SPECIFIC
      Ack : Bool;   // Сброс Аварий
      ErrorOC : Bool;   // Признак аварии по закрытию или открытию
      ErrorPower : Bool;   // Признак аварии питания
      ErrorDis : Bool;   // Признак внешней блокировки
      Error : Bool;   // Признак наличия сборной ошибки
      qON : Bool;   // Выход для управления механизмом
      closed : Bool;
      opened : Bool;
      closing : Bool;
      opening : Bool;
      errOpen : Bool;
      errClose : Bool;
      timerOpening { S7_SetPoint := 'True'} : TON_TIME;
      timerClosing { S7_SetPoint := 'True'} : TON_TIME;
      tClose : Time;
      tOpen : Time;
   END_VAR
   VAR
      AvAckAlarm_Instance { S7_SetPoint := 'True'} : "AvAckAlarm";
   END_VAR
   VAR_TEMP
      tmpDInt : DInt;
   END_VAR
   VAR_TEMP   // added for the SCL form of the ladder/FBD networks
      _w1 : Bool;
   END_VAR
BEGIN

REGION Network 1: Сброс состояния
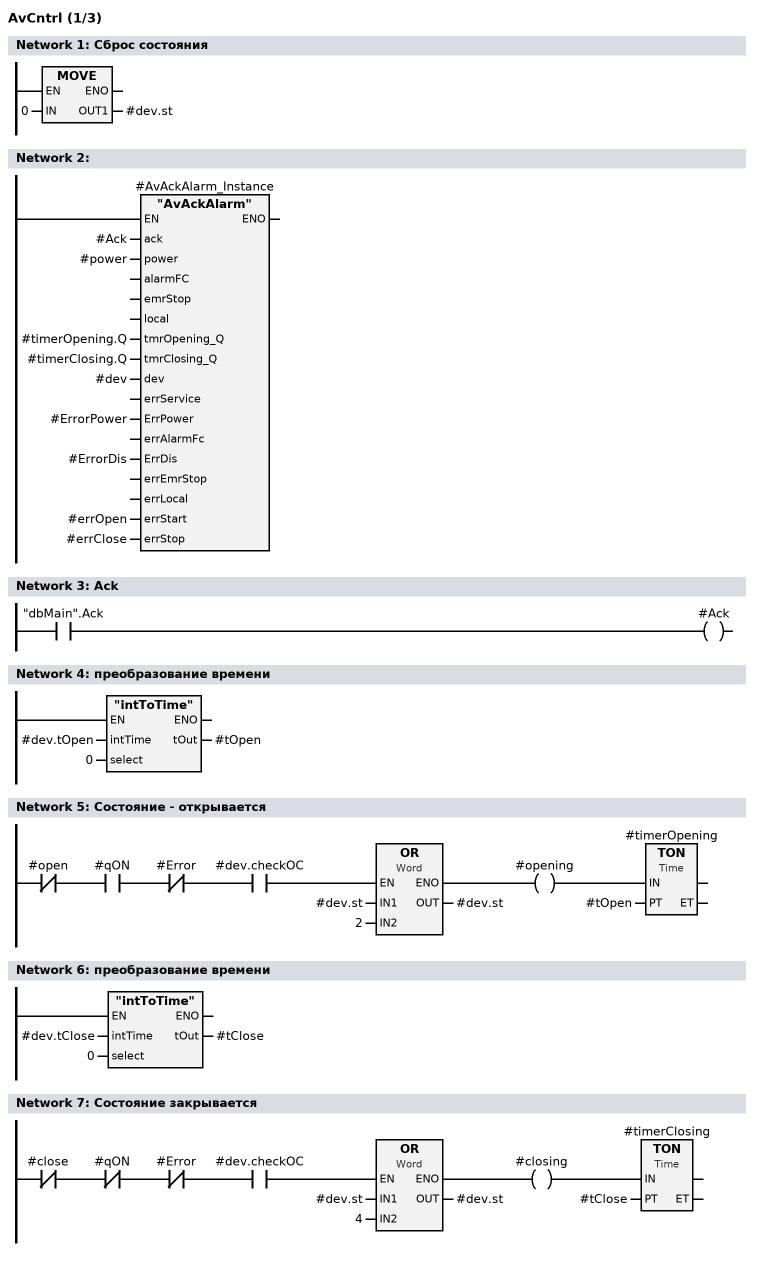
   RUNG wire#powerrail
      { S7_GenerateENO := "TRUE" } Move(in := 0, out1 => #dev.st)
   END_RUNG
   // the same network as SCL:
   #dev.st := 0;
END_REGION

REGION Network 2
   RUNG wire#powerrail
      #AvAckAlarm_Instance(ack := #Ack, power := #power, alarmFC :=, emrStop :=, local :=, tmrOpening_Q := #timerOpening.Q, tmrClosing_Q := #timerClosing.Q, dev := #dev, errService :=, ErrPower := #ErrorPower, errAlarmFc :=, ErrDis := #ErrorDis, errEmrStop :=, errLocal :=, errStart := #errOpen, errStop := #errClose)
   END_RUNG
   // the same network as SCL:
   #AvAckAlarm_Instance(ack := #Ack,   // "AvAckAlarm"
                        power := #power,
                        tmrOpening_Q := #timerOpening.Q,
                        tmrClosing_Q := #timerClosing.Q,
                        dev := #dev,
                        ErrPower := #ErrorPower,
                        ErrDis := #ErrorDis,
                        errStart := #errOpen,
                        errStop := #errClose);
END_REGION

REGION Network 3: Ack
   RUNG wire#powerrail
      Contact( "dbMain".Ack )
      Coil( #Ack )
   END_RUNG
   // the same network as SCL:
   #Ack := "dbMain".Ack;
END_REGION

REGION Network 4: преобразование времени
   RUNG wire#powerrail
      "intToTime"(intTime := #dev.tOpen, select := 0, tOut => #tOpen)
   END_RUNG
   // the same network as SCL:
   "intToTime"(intTime := #dev.tOpen, select := 0, tOut => #tOpen);
END_REGION

REGION Network 5: Состояние - открывается
   #_w1 := NOT #open AND #qON AND NOT #Error AND #dev.checkOC;
   IF #_w1 THEN #dev.st := #dev.st OR 2; END_IF;
   #opening := #_w1;
   #timerOpening(IN := #_w1, PT := #tOpen);   // TON
END_REGION

REGION Network 6: преобразование времени
   RUNG wire#powerrail
      "intToTime"(intTime := #dev.tClose, select := 0, tOut => #tClose)
   END_RUNG
   // the same network as SCL:
   "intToTime"(intTime := #dev.tClose, select := 0, tOut => #tClose);
END_REGION

REGION Network 7: Состояние закрывается
   #_w1 := NOT #close AND NOT #qON AND NOT #Error AND #dev.checkOC;
   IF #_w1 THEN #dev.st := #dev.st OR 4; END_IF;
   #closing := #_w1;
   #timerClosing(IN := #_w1, PT := #tClose);   // TON
END_REGION

REGION Network 8: Признак аварии по закрытию или открытию
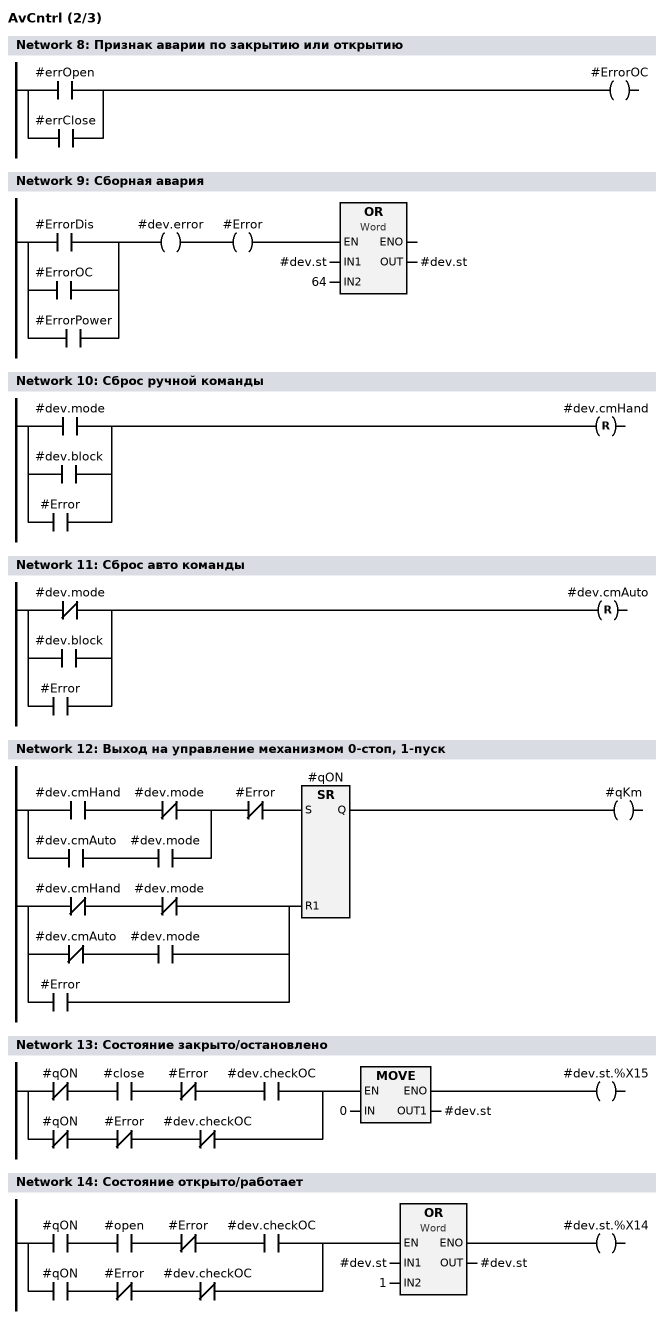
   RUNG wire#powerrail
      Contact( #errOpen )
      wire#w1
      Coil( #ErrorOC )
   END_RUNG
   RUNG wire#powerrail
      Contact( #errClose )
   END_RUNG wire#w1
   // the same network as SCL:
   #ErrorOC := #errOpen OR #errClose;
END_REGION

REGION Network 9: Сборная авария
   #dev.error := #ErrorDis OR #ErrorOC OR #ErrorPower;
   #Error := #dev.error;
   IF #dev.error THEN #dev.st := #dev.st OR 64; END_IF;
END_REGION

REGION Network 10: Сброс ручной команды
   RUNG wire#powerrail
      Contact( #dev.mode )
      wire#w1
      R_Coil( #dev.cmHand )
   END_RUNG
   RUNG wire#powerrail
      Contact( #dev.block )
   END_RUNG wire#w1
   RUNG wire#powerrail
      Contact( #Error )
   END_RUNG wire#w1
   // the same network as SCL:
   IF #dev.mode OR #dev.block OR #Error THEN #dev.cmHand := FALSE; END_IF;
END_REGION

REGION Network 11: Сброс авто команды
   RUNG wire#powerrail
      I_Contact( #dev.mode )
      wire#w1
      R_Coil( #dev.cmAuto )
   END_RUNG
   RUNG wire#powerrail
      Contact( #dev.block )
   END_RUNG wire#w1
   RUNG wire#powerrail
      Contact( #Error )
   END_RUNG wire#w1
   // the same network as SCL:
   IF NOT #dev.mode OR #dev.block OR #Error THEN #dev.cmAuto := FALSE; END_IF;
END_REGION

REGION Network 12: Выход на управление механизмом 0-стоп, 1-пуск
   RUNG wire#powerrail
      Contact( #dev.cmHand )
      I_Contact( #dev.mode )
      wire#w1
      I_Contact( #Error )
      S_SR(operand := #qON, r1 := wire#w2)
      Coil( #qKm )
   END_RUNG
   RUNG wire#powerrail
      Contact( #dev.cmAuto )
      Contact( #dev.mode )
   END_RUNG wire#w1
   RUNG wire#powerrail
      I_Contact( #dev.cmHand )
      I_Contact( #dev.mode )
   END_RUNG wire#w2
   RUNG wire#powerrail
      I_Contact( #dev.cmAuto )
      Contact( #dev.mode )
   END_RUNG wire#w2
   RUNG wire#powerrail
      Contact( #Error )
   END_RUNG wire#w2
   // the same network as SCL:
   IF ((#dev.cmHand AND NOT #dev.mode) OR (#dev.cmAuto AND #dev.mode)) AND NOT #Error THEN
       #qON := TRUE;   // SR flip-flop
   END_IF;
   IF (NOT #dev.cmHand AND NOT #dev.mode) OR (NOT #dev.cmAuto AND #dev.mode) OR #Error THEN
       #qON := FALSE;
   END_IF;
   #qKm := #qON;
END_REGION

REGION Network 13: Состояние закрыто/остановлено
   RUNG wire#powerrail
      I_Contact( #qON )
      Contact( #close )
      I_Contact( #Error )
      Contact( #dev.checkOC )
      wire#w1
      { S7_GenerateENO := "TRUE" } Move(in := 0, out1 => #dev.st)
      Coil( #dev.st.%X15 )
   END_RUNG
   RUNG wire#powerrail
      I_Contact( #qON )
      I_Contact( #Error )
      I_Contact( #dev.checkOC )
   END_RUNG wire#w1
   // the same network as SCL:
   // ENO of a box is taken as its EN; it also drops when the box reports an error
   #_w1 := (NOT #qON AND #close AND NOT #Error AND #dev.checkOC) OR (NOT #qON AND NOT #Error AND NOT #dev.checkOC);
   IF #_w1 THEN #dev.st := 0; END_IF;
   #dev.st.%X15 := #_w1;
END_REGION

REGION Network 14: Состояние открыто/работает
   #_w1 := (#qON AND #open AND NOT #Error AND #dev.checkOC) OR (#qON AND NOT #Error AND NOT #dev.checkOC);
   IF #_w1 THEN #dev.st := #dev.st OR 1; END_IF;
   #dev.st.%X14 := #_w1;
END_REGION

REGION Network 15: рУЧНОЙ режим для состояния
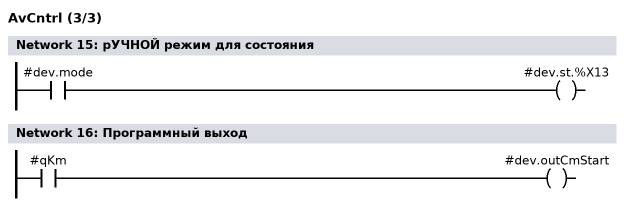
   RUNG wire#powerrail
      Contact( #dev.mode )
      Coil( #dev.st.%X13 )
   END_RUNG
   // the same network as SCL:
   #dev.st.%X13 := #dev.mode;
END_REGION

REGION Network 16: Программный выход
   RUNG wire#powerrail
      Contact( #qKm )
      Coil( #dev.outCmStart )
   END_RUNG
   // the same network as SCL:
   #dev.outCmStart := #qKm;
END_REGION
END_FUNCTION_BLOCK

FUNCTION_BLOCK "Sequencer"
{ S7_Optimized_Access := 'FALSE' }
VERSION : 0.1
   VAR_OUTPUT 
      Dev1 : Bool;
      Dev2 : Bool;
      Dev3 : Bool;
      Dev4 : Bool;
      Dev5 : Bool;
      Dev6 : Bool;
      Dev7 : Bool;
      Dev8 : Bool;
      Dev9 : Bool;
      Dev10 : Bool;
      Dev11 : Bool;
      Dev12 : Bool;
      Dev13 : Bool;
      Dev14 : Bool;
      Dev15 : Bool;
      Dev16 : Bool;
      CurTime : Time;
   END_VAR

   VAR 
      Enable : Bool;
      Hold : Bool;
      Seq : "Sequence";
      RstStep { S7_SetPoint := 'True'} : Bool := TRUE;
      Step : Int := "MIN_STEP_NUMB";
      Timer_IN { ExternalAccessible := 'False'; ExternalVisible := 'False'; ExternalWritable := 'False'} : Bool;
      Done : Bool;
      tmr : "TON_200ms";
   END_VAR

   VAR_TEMP 
      tAddStep : Bool;
   END_VAR


BEGIN
	// Управление 16-ю механизмами в зависимости 
	// от заданной последовательности Seq 
	
	IF #RstStep THEN
	    #Step := "MIN_STEP_NUMB";
	    #Timer_IN := FALSE;
	    #Done := FALSE;
	    #RstStep := FALSE;
	END_IF;
	
	#tmr(In := #Timer_IN,
	     PT := "intToTime_1"(intTime := #Seq.delay[#Step], select := 0));
	
	#Timer_IN := #Enable AND (NOT (#tmr.Q OR #Hold OR #Done));
	#CurTime := #tmr.PT - #tmr.ET;
	
	//Переход к след. шагу
	IF #tmr.Q AND (NOT #Hold) AND (NOT #Done) THEN
	    #Step += 1;
	END_IF;
	
	IF #Enable THEN //Пропуск шагов с нулевой задержкой
	    WHILE #Seq.delay[#Step] <= 0 DO
	        IF #Step >= "MAX_STEP_NUMB" THEN
	            EXIT;
	        END_IF;
	       #Step += 1;
	    END_WHILE;
	END_IF;
	
	
	//Конец последовательности
	IF #Step >= "MAX_STEP_NUMB" THEN
	    #Done := #Enable;
	    RETURN;
	END_IF;
	
	IF #Enable THEN
	    #Dev1 := #Seq.devOn[#Step, 1];
	    #Dev2 := #Seq.devOn[#Step, 2];
	    #Dev3 := #Seq.devOn[#Step, 3];
	    #Dev4 := #Seq.devOn[#Step, 4];
	    #Dev5 := #Seq.devOn[#Step, 5];
	    #Dev6 := #Seq.devOn[#Step, 6];
	    #Dev7 := #Seq.devOn[#Step, 7];
	    #Dev8 := #Seq.devOn[#Step, 8];
	    #Dev9 := #Seq.devOn[#Step, 9];
	    #Dev10 := #Seq.devOn[#Step, 10];
	    #Dev11 := #Seq.devOn[#Step, 11];
	    #Dev12 := #Seq.devOn[#Step, 12];
	    #Dev13 := #Seq.devOn[#Step, 13];
	    #Dev14 := #Seq.devOn[#Step, 14];
	    #Dev15 := #Seq.devOn[#Step, 15];
	    #Dev16 := #Seq.devOn[#Step, 16];
	END_IF;
	
	
	
	
END_FUNCTION_BLOCK

FUNCTION "intToTime_1" : Time
{ S7_Optimized_Access := 'TRUE' }
VERSION : 0.1
   VAR_INPUT 
      intTime : UInt;
      select : UInt;   // 0-sec, 1-min,2-hour
   END_VAR


BEGIN
	CASE #select OF
	    0:
	        #intToTime_1 := DINT_TO_TIME(UINT_TO_DINT(#intTime) * 1000);
	    1:
	        #intToTime_1 := DINT_TO_TIME(UINT_TO_DINT(#intTime) * 60000);
	    2:
	        #intToTime_1 := DINT_TO_TIME(UINT_TO_DINT(#intTime) * 3600000);
	    ELSE  // Statement section ELSE
	        #intToTime_1 := t#0s;
	END_CASE;
END_FUNCTION

FUNCTION_BLOCK "MDF_Handler"
{ S7_Optimized_Access := 'TRUE' }
VERSION : 0.1

BEGIN
END_FUNCTION_BLOCK

FUNCTION "LevelSelector" : Real
{ S7_Optimized_Access := 'TRUE' }
VERSION : 0.1
   VAR_INPUT 
      tankPar1 : "Ai";
      tankPar2 : "Ai";
      tankMode : Int;
   END_VAR

   VAR_OUTPUT 
      LL : Bool;
      HH : Bool;
   END_VAR

   VAR CONSTANT 
      TANK_1 : Int := 0;
      TANK_2 : Int := 1;
      TANK_1_AND_TANK_2 : Int := 2;
   END_VAR


BEGIN
	CASE #tankMode OF
	    #TANK_1:  
	        #LevelSelector := #tankPar1.Par;
	        #LL := #tankPar1.emMin;
	        #HH := #tankPar1.emMax;
	    #TANK_2: 
	        #LevelSelector := #tankPar2.Par;
	        #LL := #tankPar2.emMin;
	        #HH := #tankPar2.emMax;
	    ELSE 
	        #LevelSelector := (#tankPar1.Par + #tankPar2.Par) / 2;
	        #LL := #tankPar1.emMin OR #tankPar2.emMin;
	        #HH := #tankPar2.emMax OR #tankPar2.emMax;
	END_CASE;
	
	IF #LevelSelector < 0 THEN
	    #LevelSelector := 0;
	END_IF;
END_FUNCTION

FUNCTION "CalcNumDevUf" : Void
{ S7_Optimized_Access := 'TRUE' }
VERSION : 0.1
   VAR_INPUT 
      cmStart : Bool;
      nWorkDev : Int;   // количество работающих машин
      lev : Real;
      levStop1 : Real;
      levStart1 : Real;
      levStop2 : Real;
      levStart2 : Real;
   END_VAR

   VAR_OUTPUT 
      settingsError : Bool;
   END_VAR

   VAR_IN_OUT 
      nNeedWork : Int;
   END_VAR


BEGIN
	//проверка на корректоность настроек
	//стоп1>start11>stop2>start2
	IF #levStop1 > #levStart1 AND #levStart1 > #levStop2 AND #levStop2 > #levStart2 THEN
	    #settingsError := 0;
	ELSE
	    #settingsError := 1;
	    #nNeedWork := 0;
	    RETURN;
	END_IF;
	
	IF #cmStart THEN
	    CASE #nWorkDev OF
	        0:
	            IF #lev < #levStart1 THEN
	                #nNeedWork := 1;
	            END_IF;
	        1:
	            IF #lev < #levStart2 THEN
	                #nNeedWork := 2;
	            END_IF;
	            IF #lev > #levStop1 THEN
	                #nNeedWork := 0;
	            END_IF;
	        2:
	            IF #lev > #levStop2 THEN
	                #nNeedWork := 1;
	            END_IF;
	        ELSE
	            #nNeedWork := 0;
	    END_CASE;
	ELSE
	    #nNeedWork := 0;
	END_IF;
	
END_FUNCTION

FUNCTION "Flux" : Real
{ S7_Optimized_Access := 'TRUE' }
VERSION : 0.1
   VAR_INPUT 
      "inFlow(m3/h)" : Real;
      "Sfiltr(m2)" : Real;
   END_VAR


BEGIN
	IF (#"Sfiltr(m2)" <= 0) OR (#"inFlow(m3/h)" <= 0) THEN
	    #Flux := 0;
	    RETURN;
	ELSE
	    #Flux := (#"inFlow(m3/h)" * 1000.0) / #"Sfiltr(m2)";
	END_IF;
	
END_FUNCTION

FUNCTION_BLOCK "HandlerUF"
{ S7_Optimized_Access := 'TRUE' }
VERSION : 0.1
   VAR_INPUT 
      HDP : Bool;
      otherDeviceAvaible : Bool;
      otherDeviceInFiltration : Bool;
      filtrationTimeMin : UInt;
      delayHDP : UInt;
      maxNumbHW_ByHDP : UInt;
      HW_ToCEB1 : UInt;
      HW_ToCEB2 : UInt;
   END_VAR

   VAR_OUTPUT 
      inValve_1 : Bool;
      ownBwValve_2 : Bool;
      otherBwValve_3 : Bool;
      backFiltrValve_4 : Bool;
      clouseOtherOutValve_5 : Bool;
      outValve_6 : Bool;
      upDrainValve_7 : Bool;
      drainTankValve_8 : Bool;
      drainValve_9 : Bool;
      airValve_10 : Bool;
      filtrPump_11 : Bool;
      acidDPump_12 : Bool;
      clDPump_13 : Bool;
   END_VAR

   VAR_IN_OUT 
      flagUF : "UF_FLAGS";
      counters : "UF_COUNTERS";
      bUF : "UF_COMMANDS";
      SoftStopSeq : "Sequence";
   END_VAR

   VAR 
      cmUF : Int;
      needSoftStop : Bool;
      needHW : Bool;
      needCEB1 : Bool;
      needCEB2 : Bool;
      CEB1_ByHDP : Bool;
      CEB2_ByHDP : Bool;
      alarmHDP : Bool;
      seq : "Sequencer";
      filtration : "TONR_200ms";
      tmrHDP : "TON_200ms";
   END_VAR

   VAR_TEMP 
      i : Int;
      j : Int;
      tCmUF : Int;
      tRstFiltration : Bool;
      tHoldBW : Bool;
   END_VAR


BEGIN
	REGION Action before sequence
	    CASE #cmUF OF
	        "UF_CM_STANDBY":
	            IF NOT (#flagUF.StandBy)
	            THEN
	                "RST_UF_FLAGS"(#flagUF);
	                #flagUF.StandBy := TRUE;
	                #seq.Enable := FALSE;
	                #seq.RstStep := TRUE;
	            END_IF;
	        "UF_CM_START":
	            #seq.Seq := "dtUfSeq".START;
	            IF NOT (#flagUF.Start)
	            THEN
	                "RST_UF_FLAGS"(#flagUF);
	                #flagUF.Start := TRUE;
	                #seq.Enable := TRUE;
	                #seq.RstStep := TRUE;
	            END_IF;
	        "UF_CM_FILTRATION":
	            IF NOT (#flagUF.Filtration)
	            THEN
	                "RST_UF_FLAGS"(#flagUF);
	                #flagUF.Filtration := TRUE;
	                #seq.Enable := FALSE;
	                #seq.Done := FALSE;
	            END_IF;
	        "UF_CM_STOP":
	            IF #needSoftStop THEN
	                #seq.Seq := #SoftStopSeq;
	            ELSE
	                #seq.Seq := "dtUfSeq".STOP;
	            END_IF;
	            IF NOT (#flagUF.Stop)
	            THEN
	                "RST_UF_FLAGS"(#flagUF);
	                #flagUF.Stop := TRUE;
	                #seq.Enable := TRUE;
	                #seq.RstStep := TRUE;
	            END_IF;
	        "UF_CM_HW":
	            #seq.Seq := "dtUfSeq".HW;
	            IF NOT (#flagUF.HW) THEN
	                IF NOT(#bUF.HW) THEN
	                    "RST_UF_FLAGS"(#flagUF);
	                    #flagUF.HW := TRUE;
	                    #seq.Enable := TRUE;
	                    #seq.RstStep := TRUE;
	                    #tRstFiltration := TRUE;
	                END_IF;
	            END_IF;
	        "UF_CM_HW_A":
	            #seq.Seq := "dtUfSeq".HW_A;
	            IF NOT (#flagUF.HW_A) THEN
	                IF NOT(#bUF.HW) THEN
	                    "RST_UF_FLAGS"(#flagUF);
	                    #flagUF.HW_A := TRUE;
	                    #seq.Enable := TRUE;
	                    #seq.RstStep := TRUE;
	                    #tRstFiltration := TRUE;
	                END_IF;
	            END_IF;
	        "UF_CM_CEB1":
	            #seq.Seq := "dtUfSeq".CEB1;
	            IF NOT (#flagUF.CEB1) THEN
	                IF NOT(#flagUF.CEB1) THEN
	                    "RST_UF_FLAGS"(#flagUF);
	                    #flagUF.CEB1 := TRUE;
	                    #seq.Enable := TRUE;
	                    #seq.RstStep := TRUE;
	                    #tRstFiltration := TRUE;
	                END_IF;
	            END_IF;
	        "UF_CM_CEB1_A":
	            #seq.Seq := "dtUfSeq".CEB1_A;
	            IF NOT (#flagUF.CEB1_A) THEN
	                IF NOT(#flagUF.CEB1_A) THEN
	                    "RST_UF_FLAGS"(#flagUF);
	                    #flagUF.CEB1_A := TRUE;
	                    #seq.Enable := TRUE;
	                    #seq.RstStep := TRUE;
	                    #tRstFiltration := TRUE;
	                END_IF;
	            END_IF;
	        "UF_CM_CEB2":
	            #seq.Seq := "dtUfSeq".CEB2;
	            IF NOT (#flagUF.CEB2) THEN
	                IF NOT (#flagUF.CEB1) THEN
	                    "RST_UF_FLAGS"(#flagUF);
	                    #flagUF.CEB2 := TRUE;
	                    #seq.Enable := TRUE;
	                    #seq.RstStep := TRUE;
	                    #tRstFiltration := TRUE;
	                END_IF;
	            END_IF;
	        "UF_CM_CEB2_A":
	            #seq.Seq := "dtUfSeq".CEB2_A;
	            IF NOT (#flagUF.CEB2_A) THEN
	                IF NOT (#flagUF.CEB2_A) THEN
	                    "RST_UF_FLAGS"(#flagUF);
	                    #flagUF.CEB2_A := TRUE;
	                    #seq.Enable := TRUE;
	                    #seq.RstStep := TRUE;
	                    #tRstFiltration := TRUE;
	                END_IF;
	
	            END_IF;
	    END_CASE;
	END_REGION
	REGION Soft stop HW, CEB1, CEB2 (if wash was interrupt by dissable other UF)
	    CASE #cmUF OF
	        "UF_CM_HW",
	        "UF_CM_CEB1",
	        "UF_CM_CEB2":
	            IF NOT (#otherDeviceAvaible) THEN
	                #cmUF := "UF_CM_STOP";
	                #needSoftStop := TRUE;
	                //Build sequence
	                FOR #i := "MIN_STEP_NUMB" TO 5 DO
	                    CASE #i OF
	                        1:  // Turn off pumps
	                            #SoftStopSeq.devOn[#i] := #seq.Seq.devOn[#seq.Step];
	                            #SoftStopSeq.devOn[#i, 11] := FALSE; //filtrate pump 
	                            #SoftStopSeq.devOn[#i, 12] := FALSE; //acid
	                            #SoftStopSeq.devOn[#i, 13] := FALSE; //clorine
	                            #SoftStopSeq.devOn[#i + 1] := #SoftStopSeq.devOn[#i];
	                        2: // Clouse in valves.
	                            #SoftStopSeq.devOn[#i, 1] := FALSE; //in valve
	                            #SoftStopSeq.devOn[#i, 4] := FALSE; //back filtrate valve.
	                            #SoftStopSeq.devOn[#i, 5] := FALSE; //Turn off command to clouse other UF out valve
	                            #SoftStopSeq.devOn[#i, 10] := FALSE; //air
	                            #SoftStopSeq.devOn[#i + 1] := #SoftStopSeq.devOn[#i];
	                        3: //Clouse valves...
	                            #SoftStopSeq.devOn[#i, 2] := FALSE; //own bw
	                            #SoftStopSeq.devOn[#i, 3] := FALSE; //other bw
	                            #SoftStopSeq.devOn[#i, 6] := FALSE; //out
	                            #SoftStopSeq.devOn[#i, 8] := FALSE; //drain to tank
	                            #SoftStopSeq.devOn[#i + 1] := #SoftStopSeq.devOn[#i];
	                        4: //Clouse valves...
	                            #SoftStopSeq.devOn[#i, 9] := FALSE; //drain
	                            #SoftStopSeq.devOn[#i, 7] := FALSE; //up drain
	                        5: //Turn off all
	                            #SoftStopSeq.devOn[#i, 1] :=
	                            #SoftStopSeq.devOn[#i, 2] :=
	                            #SoftStopSeq.devOn[#i, 3] :=
	                            #SoftStopSeq.devOn[#i, 4] :=
	                            #SoftStopSeq.devOn[#i, 5] :=
	                            #SoftStopSeq.devOn[#i, 6] :=
	                            #SoftStopSeq.devOn[#i, 7] :=
	                            #SoftStopSeq.devOn[#i, 8] :=
	                            #SoftStopSeq.devOn[#i, 9] :=
	                            #SoftStopSeq.devOn[#i, 10] :=
	                            #SoftStopSeq.devOn[#i, 11] :=
	                            #SoftStopSeq.devOn[#i, 12] :=
	                            #SoftStopSeq.devOn[#i, 13] :=
	                            #SoftStopSeq.devOn[#i, 14] :=
	                            #SoftStopSeq.devOn[#i, 15] :=
	                            #SoftStopSeq.devOn[#i, 16] := FALSE;
	                    END_CASE;
	                END_FOR;
	            END_IF;
	    END_CASE;
	END_REGION
	REGION High preassure difference
	    #tmrHDP(In := #flagUF.Filtration AND #HDP,
	            PT := "intToTime_1"(intTime := #delayHDP, select := 0));
	END_REGION
	REGION Filtration
	    #filtration(In := #flagUF.Filtration,
	                PT := "intToTime_1"(intTime := #filtrationTimeMin, select := 0),
	                R := #tRstFiltration);
	END_REGION
	REGION Hold sequencer
	    #tHoldBW := #ownBwValve_2 AND #flagUF.HW AND NOT(#otherDeviceInFiltration);
	    #seq.Hold := #tHoldBW;
	END_REGION
	REGION Sequencer
	    #seq(Dev1 => #inValve_1,
	         Dev2 => #ownBwValve_2,
	         Dev3 => #otherBwValve_3,
	         Dev4 => #backFiltrValve_4,
	         Dev5 => #clouseOtherOutValve_5,
	         Dev6 => #outValve_6,
	         Dev7 => #upDrainValve_7,
	         Dev8 => #drainTankValve_8,
	         Dev9 => #drainValve_9,
	         Dev10 => #airValve_10,
	         Dev11 => #filtrPump_11,
	         Dev12 => #acidDPump_12,
	         Dev13 => #clDPump_13);
	END_REGION
	REGION Action after sequence done
	    IF #seq.Done OR #filtration.Q OR #tmrHDP.Q THEN
	      #tCmUF := #cmUF;
	      CASE #cmUF OF
	          "UF_CM_STANDBY": // After standby -> nothing
	              ;
	          "UF_CM_START": //After start -> filtration
	              #tCmUF := "UF_CM_FILTRATION";
	          "UF_CM_FILTRATION": //After filtration...
	              IF #otherDeviceAvaible THEN //Permition for stop
	                  IF NOT (#bUF.HW OR #bUF.CEB1 OR #bUF.CEB2) THEN //Simple HW
	                      #tCmUF := "UF_CM_STOP";
	                  END_IF;
	              ELSE
	                  IF NOT (#bUF.HW_A OR #bUF.CEB1_A OR #bUF.CEB2_A) THEN // Custom HW
	                      #tCmUF := "UF_CM_STOP";
	                  END_IF;
	              END_IF;
	              IF #tCmUF = "UF_CM_STOP" THEN // only after permition
	                  IF #filtration.Q THEN //Filtration done...
	                      #counters.HDPW := 0; //RST HDP counters and flags
	                      #CEB1_ByHDP := #CEB2_ByHDP := FALSE;
	                      IF #counters.HW >= #HW_ToCEB2 THEN // -> CEB2
	                          #needCEB2 := TRUE;
	                      ELSIF #counters.HW = (#HW_ToCEB1 * (#counters.CEB1 + 1)) THEN // -> CEB1
	                          #needCEB1 := TRUE;
	                      ELSE // -> HW
	                          #needHW := TRUE;
	                      END_IF;
	                  END_IF;
	                  IF #tmrHDP.Q THEN //When high delta preassure -> HW -> max count of HW -> CEB1 -> CEB2 -> alarm
	                    #counters.HDPW += 1;
	                    IF #counters.HDPW <= #maxNumbHW_ByHDP THEN
	                        #needHW := TRUE;
	                    ELSE
	                        IF #CEB1_ByHDP THEN //Do CEB1 when counter more then max number
	                              IF #CEB2_ByHDP THEN //Do CEB2 after CEB1; Again CEB2 by HDP -> alarm
	                                #alarmHDP := TRUE;
	                            ELSE
	                                #CEB2_ByHDP := TRUE;
	                                #needCEB2 := TRUE;
	                            END_IF;
	                        ELSE
	                            #CEB1_ByHDP := TRUE;
	                            #needCEB1 := TRUE;
	                        END_IF;
	                    END_IF;
	                END_IF;
	            END_IF;
	          "UF_CM_STOP": //Stop...
	              #needSoftStop := FALSE;
	             IF #alarmHDP THEN //by HDP alarm -> standby
	                #tCmUF := "UF_CM_STANDBY";
	                #alarmHDP :=
	//                #needHW :=
	//                #needCEB1 :=
	//                #needCEB2 :=
	                #CEB1_ByHDP := 
	                #CEB2_ByHDP := FALSE;
	                #counters.HDPW := 0;
	                #flagUF.ErrHDP := TRUE;
	            ELSIF #needHW THEN //by request HW -> HW/HW_A
	                #counters.HW += 1;
	                IF #otherDeviceAvaible THEN
	                    #tCmUF := "UF_CM_HW";
	                ELSE
	                    #tCmUF := "UF_CM_HW_A";
	                END_IF;
	            ELSIF #needCEB1 THEN //by request CEB1 -> CEB1/CEB1_A
	                #counters.CEB1 += 1;
	                IF #otherDeviceAvaible THEN
	                    #tCmUF := "UF_CM_CEB1";
	                ELSE
	                    #tCmUF := "UF_CM_CEB1_A";
	                END_IF;
	            ELSIF #needCEB2 THEN //by request CEB2 -> CEB2/CEB2_A
	                #counters.HW := #counters.CEB1 := 0;
	                #counters.CEB2 += 1;
	                IF #otherDeviceAvaible THEN
	                    #tCmUF := "UF_CM_CEB2";
	                ELSE
	                    #tCmUF := "UF_CM_CEB2_A";
	                END_IF;
	            ELSE //simple stop -> standby
	                #tCmUF := "UF_CM_STANDBY";
	            END_IF;
	          "UF_CM_HW",
	          "UF_CM_HW_A": //HW -> Standby
	              #needHW := FALSE;
	              #tCmUF := "UF_CM_STANDBY";
	          "UF_CM_CEB1",
	          "UF_CM_CEB1_A": //CEB1 -> Standby
	              #needCEB1 := FALSE;
	              #tCmUF := "UF_CM_STANDBY";
	          "UF_CM_CEB2",
	          "UF_CM_CEB2_A": //CEB2 -> Standby
	              #needCEB2 := FALSE;
	              #tCmUF := "UF_CM_STANDBY";
	      END_CASE;
	      #cmUF := #tCmUF;
	    END_IF;
	END_REGION
	REGION Error flag
	    #flagUF.Err :=
	    #flagUF.ErrWork
	    OR #flagUF.ErrHW
	    OR #flagUF.ErrCEB1
	    OR #flagUF.ErrCEB2
	    OR #flagUF.ErrHDP;
	END_REGION
	
	  
END_FUNCTION_BLOCK

DATA_BLOCK "hardwareTimePulse_DB"   // DB13
VERSION : 0.1
// stored: AutoNumber true, DBAccessibleFromOPCUA true, InstanceOfName hardwareTimePulse, InstanceOfType FB
"hardwareTimePulse"
BEGIN
END_DATA_BLOCK

DATA_BLOCK "AllDpump_DB"   // DB27
VERSION : 0.1
// stored: AutoNumber true, DBAccessibleFromOPCUA true, InstanceOfName AllDpump, InstanceOfType FB
"AllDpump"
   // VAR
   //    dp101 { S7_SetPoint := 'True'} : "DPumpCntr";
   //    dp501 { S7_SetPoint := 'True'} : "DPumpCntr";
   //    dp502 { S7_SetPoint := 'True'} : "DPumpCntr";
   //    dp801 { S7_SetPoint := 'True'} : "DPumpCntr";
   //    dp802 { S7_SetPoint := 'True'} : "DPumpCntr";
   //    dp803 { S7_SetPoint := 'True'} : "DPumpCntr";
   //    dp1001 { S7_SetPoint := 'True'} : "DPumpCntr";
   // END_VAR
BEGIN
END_DATA_BLOCK

DATA_BLOCK "AllDigital_DB"   // DB17
VERSION : 0.1
// stored: AutoNumber true, DBAccessibleFromOPCUA true, InstanceOfName AllDigital, InstanceOfType FB
"AllDigital"
BEGIN
END_DATA_BLOCK

DATA_BLOCK "AllFlowCounter_DB"   // DB29
VERSION : 0.1
// stored: AutoNumber true, DBAccessibleFromOPCUA true, InstanceOfName AllFlowCounter, InstanceOfType FB
"AllFlowCounter"
BEGIN
END_DATA_BLOCK

DATA_BLOCK "AllPID_DB"   // DB11
VERSION : 0.1
// stored: AutoNumber true, DBAccessibleFromOPCUA true, InstanceOfName AllPID, InstanceOfType FB
"AllPID"
BEGIN
END_DATA_BLOCK

DATA_BLOCK "AllPump_DB"   // DB9
VERSION : 0.1
// stored: AutoNumber true, DBAccessibleFromOPCUA true, InstanceOfName AllPump, InstanceOfType FB
"AllPump"
BEGIN
END_DATA_BLOCK

DATA_BLOCK "AllUF_DB"   // DB28
VERSION : 0.1
// stored: AutoNumber true, DBAccessibleFromOPCUA true, InstanceOfName AllUF, InstanceOfType FB
"AllUF"
   // VAR
   //    reqNumbWorkUF { ExternalVisible := 'False'; ExternalWritable := 'False'} : USInt;
   //    readyUF : Array[0..1] of Bool;
   //    workUF : Array[0..1] of Bool;
   //    cmUF : Array[0..1] of Bool;
   //    HandlerUF1 { S7_SetPoint := 'True'} : "HandlerUF";
   //    HandlerUF2 { S7_SetPoint := 'True'} : "HandlerUF";
   // END_VAR
BEGIN
END_DATA_BLOCK

DATA_BLOCK "AllUfParam_DB"   // DB30
VERSION : 0.1
// stored: AutoNumber true, DBAccessibleFromOPCUA true, InstanceOfName AllUfParam, InstanceOfType FB
"AllUfParam"
   // VAR
   //    mSec : USInt;
   //    sec : UInt;
   //    inVolumeUF1 : Real;
   //    inVolumeUF2 : Real;
   //    outVolumeUF1 : Real;
   //    outVolumeUF2 : Real;
   // END_VAR
BEGIN
END_DATA_BLOCK

DATA_BLOCK "AllAv_DB"   // DB3
VERSION : 0.1
// stored: AutoNumber true, DBAccessibleFromOPCUA true, InstanceOfName AllAv, InstanceOfType FB
"AllAv"
   // VAR
   //    DVM201 { S7_SetPoint := 'True'} : "AvCntrl";
   //    SOV801 { S7_SetPoint := 'True'} : "AvCntrl";
   //    SOV901 { S7_SetPoint := 'True'} : "AvCntrl";
   //    SOV902 { S7_SetPoint := 'True'} : "AvCntrl";
   //    SOV1301 { S7_SetPoint := 'True'} : "AvCntrl";
   //    SOV1302 { S7_SetPoint := 'True'} : "AvCntrl";
   //    SOV1303 { S7_SetPoint := 'True'} : "AvCntrl";
   //    DVA501 { S7_SetPoint := 'True'} : "AvCntrl";
   //    DVA502 { S7_SetPoint := 'True'} : "AvCntrl";
   //    DVA504 { S7_SetPoint := 'True'} : "AvCntrl";
   //    DVA505 { S7_SetPoint := 'True'} : "AvCntrl";
   //    DVA506 { S7_SetPoint := 'True'} : "AvCntrl";
   //    DVA507 { S7_SetPoint := 'True'} : "AvCntrl";
   //    DVA508 { S7_SetPoint := 'True'} : "AvCntrl";
   //    DVA509 { S7_SetPoint := 'True'} : "AvCntrl";
   //    DVA511 { S7_SetPoint := 'True'} : "AvCntrl";
   //    DVA512 { S7_SetPoint := 'True'} : "AvCntrl";
   //    DVA513 { S7_SetPoint := 'True'} : "AvCntrl";
   //    DVA514 { S7_SetPoint := 'True'} : "AvCntrl";
   //    DVA515 { S7_SetPoint := 'True'} : "AvCntrl";
   //    DVA516 { S7_SetPoint := 'True'} : "AvCntrl";
   //    DVA1801 { S7_SetPoint := 'True'} : "AvCntrl";
   // END_VAR
BEGIN
END_DATA_BLOCK

DATA_BLOCK "tmrAck"   // DB10
{ S7_Optimized_Access := 'TRUE' }
// stored: AutoNumber true, DBAccessibleFromOPCUA true, InstanceOfName IEC_TIMER, OfSystemLibElement IEC_TIMER, OfSystemLibVersion 1.0
"IEC_TIMER"
   // VAR
   //    PT : Time;
   //    ET { ExternalWritable := 'False'} : Time;
   //    IN : Bool;
   //    Q { ExternalWritable := 'False'} : Bool;
   // END_VAR
BEGIN
END_DATA_BLOCK
